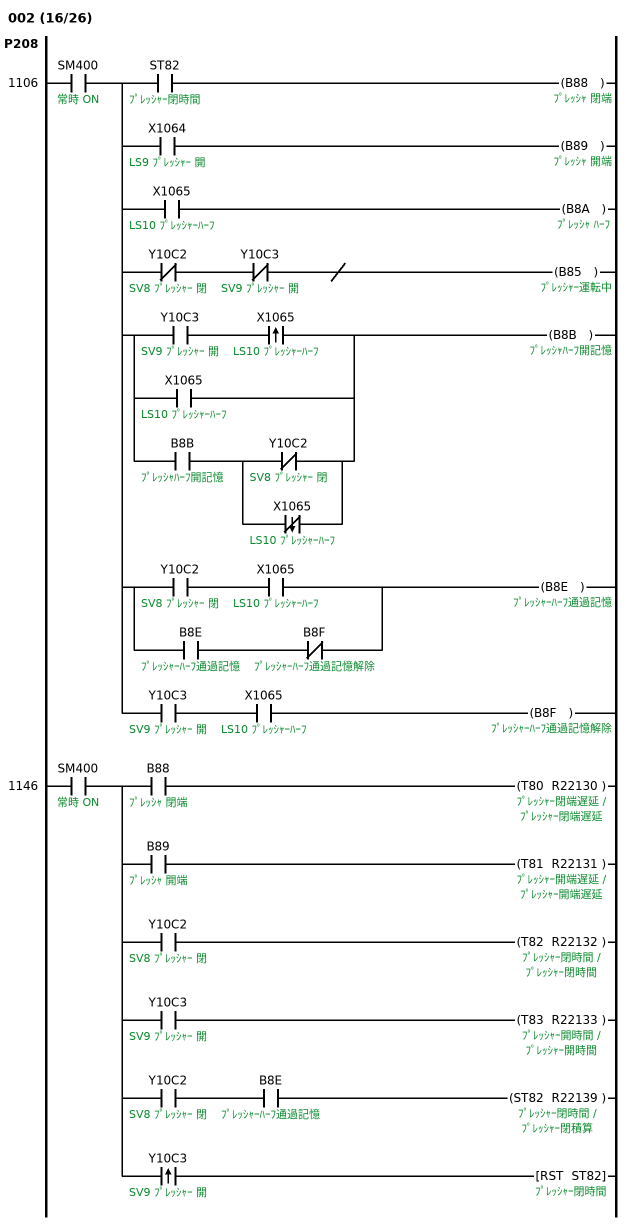
1106  LD      SM400  ; 常時 ON
      MPS
      AND     ST82  ; ﾌﾟﾚｯｼｬｰ閉時間
      OUT     B88  ; ﾌﾟﾚｯｼｬ 閉端
      MRD
      AND     X1064  ; LS9 ﾌﾟﾚｯｼｬｰ 開
      OUT     B89  ; ﾌﾟﾚｯｼｬ 開端
      MRD
      AND     X1065  ; LS10 ﾌﾟﾚｯｼｬｰﾊｰﾌ
      OUT     B8A  ; ﾌﾟﾚｯｼｬ ﾊｰﾌ
      MRD
      ANI     Y10C2  ; SV8 ﾌﾟﾚｯｼｬｰ 閉
      ANI     Y10C3  ; SV9 ﾌﾟﾚｯｼｬｰ 開
      INV
      OUT     B85  ; ﾌﾟﾚｯｼｬｰ運転中
      MRD
      LD      Y10C3  ; SV9 ﾌﾟﾚｯｼｬｰ 開
      ANDP    X1065  ; LS10 ﾌﾟﾚｯｼｬｰﾊｰﾌ
      OR      X1065  ; LS10 ﾌﾟﾚｯｼｬｰﾊｰﾌ
      LD      B8B  ; ﾌﾟﾚｯｼｬﾊｰﾌ開記憶
      LDI     Y10C2  ; SV8 ﾌﾟﾚｯｼｬｰ 閉
      ORFI    X1065  ; LS10 ﾌﾟﾚｯｼｬｰﾊｰﾌ
      ANB
      ORB
      ANB
      OUT     B8B  ; ﾌﾟﾚｯｼｬﾊｰﾌ開記憶
      MRD
      LD      Y10C2  ; SV8 ﾌﾟﾚｯｼｬｰ 閉
      AND     X1065  ; LS10 ﾌﾟﾚｯｼｬｰﾊｰﾌ
      LD      B8E  ; ﾌﾟﾚｯｼｬｰﾊｰﾌ通過記憶
      ANI     B8F  ; ﾌﾟﾚｯｼｬｰﾊｰﾌ通過記憶解除
      ORB
      ANB
      OUT     B8E  ; ﾌﾟﾚｯｼｬｰﾊｰﾌ通過記憶
      MPP
      AND     Y10C3  ; SV9 ﾌﾟﾚｯｼｬｰ 開
      AND     X1065  ; LS10 ﾌﾟﾚｯｼｬｰﾊｰﾌ
      OUT     B8F  ; ﾌﾟﾚｯｼｬｰﾊｰﾌ通過記憶解除
1146  LD      SM400  ; 常時 ON
      MPS
      AND     B88  ; ﾌﾟﾚｯｼｬ 閉端
      OUT     T80 R22130  ; ﾌﾟﾚｯｼｬｰ閉端遅延 / ﾌﾟﾚｯｼｬｰ閉端遅延
      MRD
      AND     B89  ; ﾌﾟﾚｯｼｬ 開端
      OUT     T81 R22131  ; ﾌﾟﾚｯｼｬｰ開端遅延 / ﾌﾟﾚｯｼｬｰ開端遅延
      MRD
      AND     Y10C2  ; SV8 ﾌﾟﾚｯｼｬｰ 閉
      OUT     T82 R22132  ; ﾌﾟﾚｯｼｬｰ閉時間 / ﾌﾟﾚｯｼｬｰ閉時間
      MRD
      AND     Y10C3  ; SV9 ﾌﾟﾚｯｼｬｰ 開
      OUT     T83 R22133  ; ﾌﾟﾚｯｼｬｰ開時間 / ﾌﾟﾚｯｼｬｰ開時間
      MRD
      AND     Y10C2  ; SV8 ﾌﾟﾚｯｼｬｰ 閉
      AND     B8E  ; ﾌﾟﾚｯｼｬｰﾊｰﾌ通過記憶
      OUT     ST82 R22139  ; ﾌﾟﾚｯｼｬｰ閉時間 / ﾌﾟﾚｯｼｬｰ閉積算
      MPP
      ANDP    Y10C3  ; SV9 ﾌﾟﾚｯｼｬｰ 開
      RST     ST82  ; ﾌﾟﾚｯｼｬｰ閉時間
; 
      P209
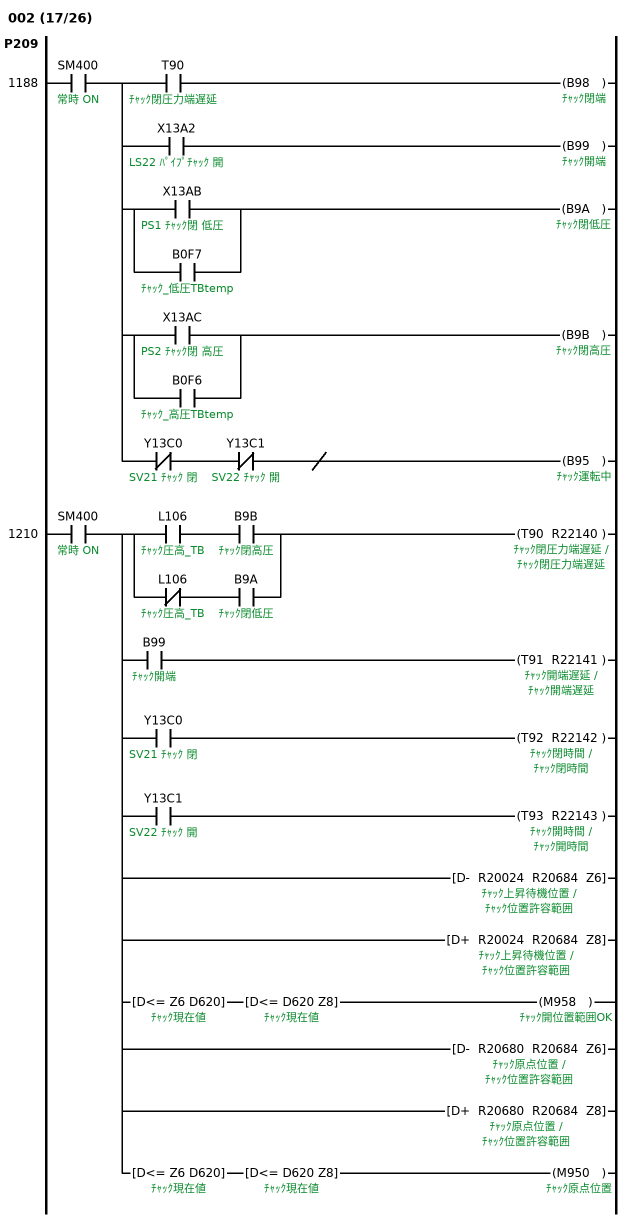
1188  LD      SM400  ; 常時 ON
      MPS
      AND     T90  ; ﾁｬｯｸ閉圧力端遅延
      OUT     B98  ; ﾁｬｯｸ閉端
      MRD
      AND     X13A2  ; LS22 ﾊﾟｲﾌﾟﾁｬｯｸ 開
      OUT     B99  ; ﾁｬｯｸ開端
      MRD
      LD      X13AB  ; PS1 ﾁｬｯｸ閉 低圧
      OR      B0F7  ; ﾁｬｯｸ_低圧TBtemp
      ANB
      OUT     B9A  ; ﾁｬｯｸ閉低圧
      MRD
      LD      X13AC  ; PS2 ﾁｬｯｸ閉 高圧
      OR      B0F6  ; ﾁｬｯｸ_高圧TBtemp
      ANB
      OUT     B9B  ; ﾁｬｯｸ閉高圧
      MPP
      ANI     Y13C0  ; SV21 ﾁｬｯｸ 閉
      ANI     Y13C1  ; SV22 ﾁｬｯｸ 開
      INV
      OUT     B95  ; ﾁｬｯｸ運転中
1210  LD      SM400  ; 常時 ON
      MPS
      LD      L106  ; ﾁｬｯｸ圧高_TB
      AND     B9B  ; ﾁｬｯｸ閉高圧
      LDI     L106  ; ﾁｬｯｸ圧高_TB
      AND     B9A  ; ﾁｬｯｸ閉低圧
      ORB
      ANB
      OUT     T90 R22140  ; ﾁｬｯｸ閉圧力端遅延 / ﾁｬｯｸ閉圧力端遅延
      MRD
      AND     B99  ; ﾁｬｯｸ開端
      OUT     T91 R22141  ; ﾁｬｯｸ開端遅延 / ﾁｬｯｸ開端遅延
      MRD
      AND     Y13C0  ; SV21 ﾁｬｯｸ 閉
      OUT     T92 R22142  ; ﾁｬｯｸ閉時間 / ﾁｬｯｸ閉時間
      MRD
      AND     Y13C1  ; SV22 ﾁｬｯｸ 開
      OUT     T93 R22143  ; ﾁｬｯｸ開時間 / ﾁｬｯｸ開時間
      MPP
      D-      R20024 R20684 Z6  ; ﾁｬｯｸ位置許容範囲
      D+      R20024 R20684 Z8
      MPS
      ANDD<=  Z6 D620  ; ﾁｬｯｸ現在値
      ANDD<=  D620 Z8  ; ﾁｬｯｸ現在値
      OUT     M958  ; ﾁｬｯｸ開位置範囲OK
      MPP
      D-      R20680 R20684 Z6  ; ﾁｬｯｸ原点位置
      D+      R20680 R20684 Z8
      ANDD<=  Z6 D620  ; ﾁｬｯｸ現在値
      ANDD<=  D620 Z8  ; ﾁｬｯｸ現在値
      OUT     M950  ; ﾁｬｯｸ原点位置
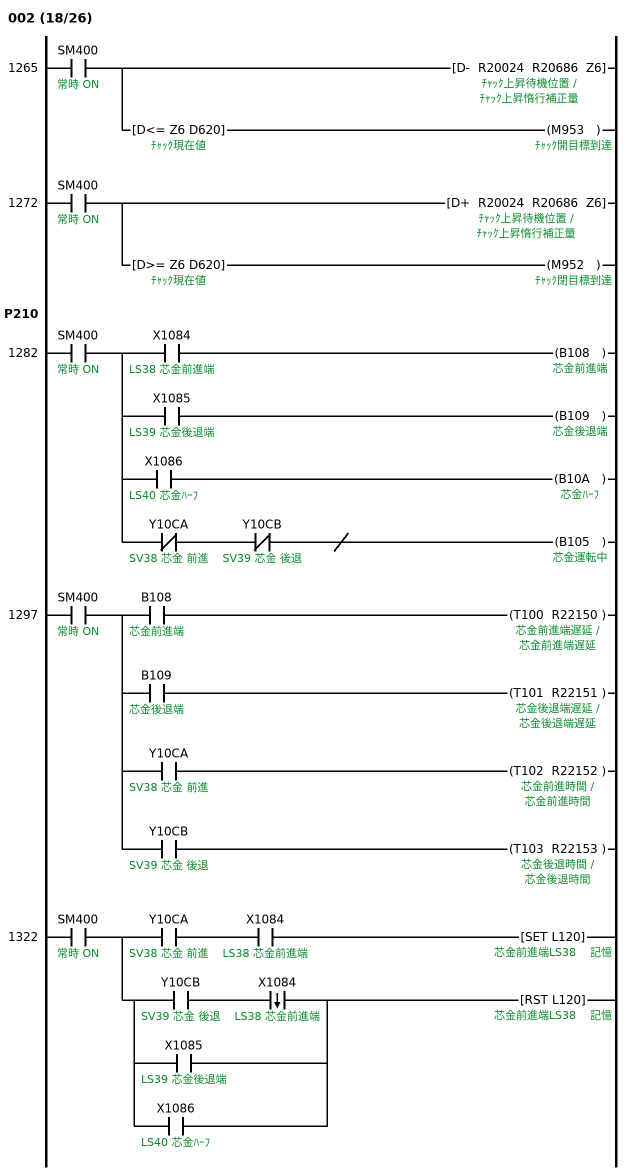
1265  LD      SM400  ; 常時 ON
      D-      R20024 R20686 Z6  ; ﾁｬｯｸ上昇惰行補正量
      ANDD<=  Z6 D620  ; ﾁｬｯｸ現在値
      OUT     M953  ; ﾁｬｯｸ開目標到達
1272  LD      SM400  ; 常時 ON
      D+      R20024 R20686 Z6
      ANDD>=  Z6 D620  ; ﾁｬｯｸ現在値
      OUT     M952  ; ﾁｬｯｸ閉目標到達
; 
      P210
1282  LD      SM400  ; 常時 ON
      MPS
      AND     X1084  ; LS38 芯金前進端
      OUT     B108  ; 芯金前進端
      MRD
      AND     X1085  ; LS39 芯金後退端
      OUT     B109  ; 芯金後退端
      MRD
      AND     X1086  ; LS40 芯金ﾊｰﾌ
      OUT     B10A  ; 芯金ﾊｰﾌ
      MPP
      ANI     Y10CA  ; SV38 芯金 前進
      ANI     Y10CB  ; SV39 芯金 後退
      INV
      OUT     B105  ; 芯金運転中
1297  LD      SM400  ; 常時 ON
      MPS
      AND     B108  ; 芯金前進端
      OUT     T100 R22150  ; 芯金前進端遅延 / 芯金前進端遅延
      MRD
      AND     B109  ; 芯金後退端
      OUT     T101 R22151  ; 芯金後退端遅延 / 芯金後退端遅延
      MRD
      AND     Y10CA  ; SV38 芯金 前進
      OUT     T102 R22152  ; 芯金前進時間 / 芯金前進時間
      MPP
      AND     Y10CB  ; SV39 芯金 後退
      OUT     T103 R22153  ; 芯金後退時間 / 芯金後退時間
1322  LD      SM400  ; 常時 ON
      MPS
      AND     Y10CA  ; SV38 芯金 前進
      AND     X1084  ; LS38 芯金前進端
      SET     L120  ; 芯金前進端LS38    記憶
      MPP
      LD      Y10CB  ; SV39 芯金 後退
      ANDF    X1084  ; LS38 芯金前進端
      OR      X1085  ; LS39 芯金後退端
      OR      X1086  ; LS40 芯金ﾊｰﾌ
      ANB
      RST     L120  ; 芯金前進端LS38    記憶
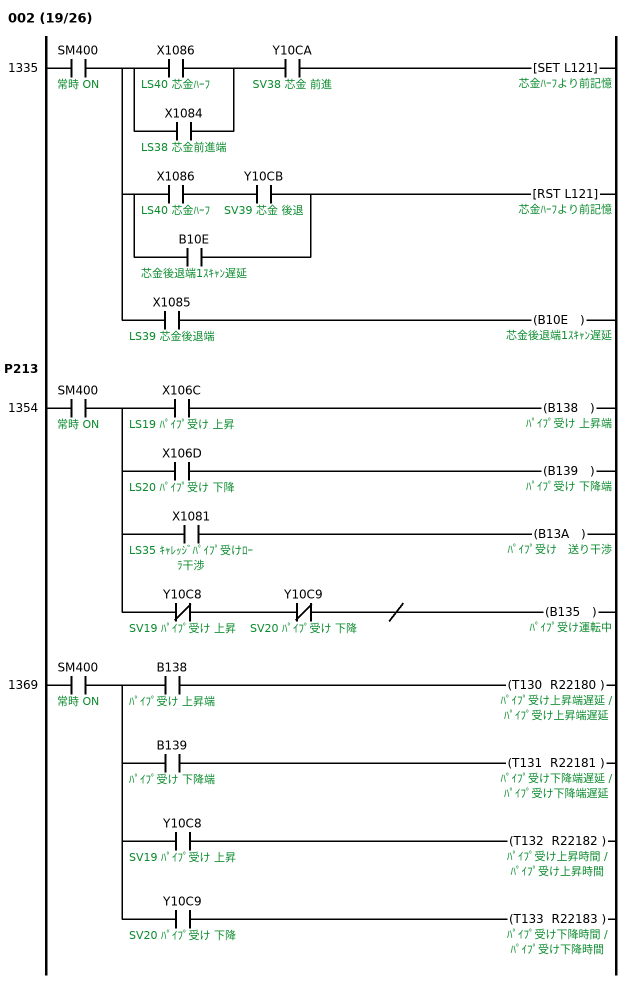
1335  LD      SM400  ; 常時 ON
      MPS
      LD      X1086  ; LS40 芯金ﾊｰﾌ
      OR      X1084  ; LS38 芯金前進端
      ANB
      AND     Y10CA  ; SV38 芯金 前進
      SET     L121  ; 芯金ﾊｰﾌより前記憶
      MRD
      LD      X1086  ; LS40 芯金ﾊｰﾌ
      AND     Y10CB  ; SV39 芯金 後退
      OR      B10E  ; 芯金後退端1ｽｷｬﾝ遅延
      ANB
      RST     L121  ; 芯金ﾊｰﾌより前記憶
      MPP
      AND     X1085  ; LS39 芯金後退端
      OUT     B10E  ; 芯金後退端1ｽｷｬﾝ遅延
; 
      P213
1354  LD      SM400  ; 常時 ON
      MPS
      AND     X106C  ; LS19 ﾊﾟｲﾌﾟ受け 上昇
      OUT     B138  ; ﾊﾟｲﾌﾟ受け 上昇端
      MRD
      AND     X106D  ; LS20 ﾊﾟｲﾌﾟ受け 下降
      OUT     B139  ; ﾊﾟｲﾌﾟ受け 下降端
      MRD
      AND     X1081  ; LS35 ｷｬﾚｯｼﾞﾊﾟｲﾌﾟ受けﾛｰﾗ干渉
      OUT     B13A  ; ﾊﾟｲﾌﾟ受け　送り干渉
      MPP
      ANI     Y10C8  ; SV19 ﾊﾟｲﾌﾟ受け 上昇
      ANI     Y10C9  ; SV20 ﾊﾟｲﾌﾟ受け 下降
      INV
      OUT     B135  ; ﾊﾟｲﾌﾟ受け運転中
1369  LD      SM400  ; 常時 ON
      MPS
      AND     B138  ; ﾊﾟｲﾌﾟ受け 上昇端
      OUT     T130 R22180  ; ﾊﾟｲﾌﾟ受け上昇端遅延 / ﾊﾟｲﾌﾟ受け上昇端遅延
      MRD
      AND     B139  ; ﾊﾟｲﾌﾟ受け 下降端
      OUT     T131 R22181  ; ﾊﾟｲﾌﾟ受け下降端遅延 / ﾊﾟｲﾌﾟ受け下降端遅延
      MRD
      AND     Y10C8  ; SV19 ﾊﾟｲﾌﾟ受け 上昇
      OUT     T132 R22182  ; ﾊﾟｲﾌﾟ受け上昇時間 / ﾊﾟｲﾌﾟ受け上昇時間
      MPP
      AND     Y10C9  ; SV20 ﾊﾟｲﾌﾟ受け 下降
      OUT     T133 R22183  ; ﾊﾟｲﾌﾟ受け下降時間 / ﾊﾟｲﾌﾟ受け下降時間
; 
      P214
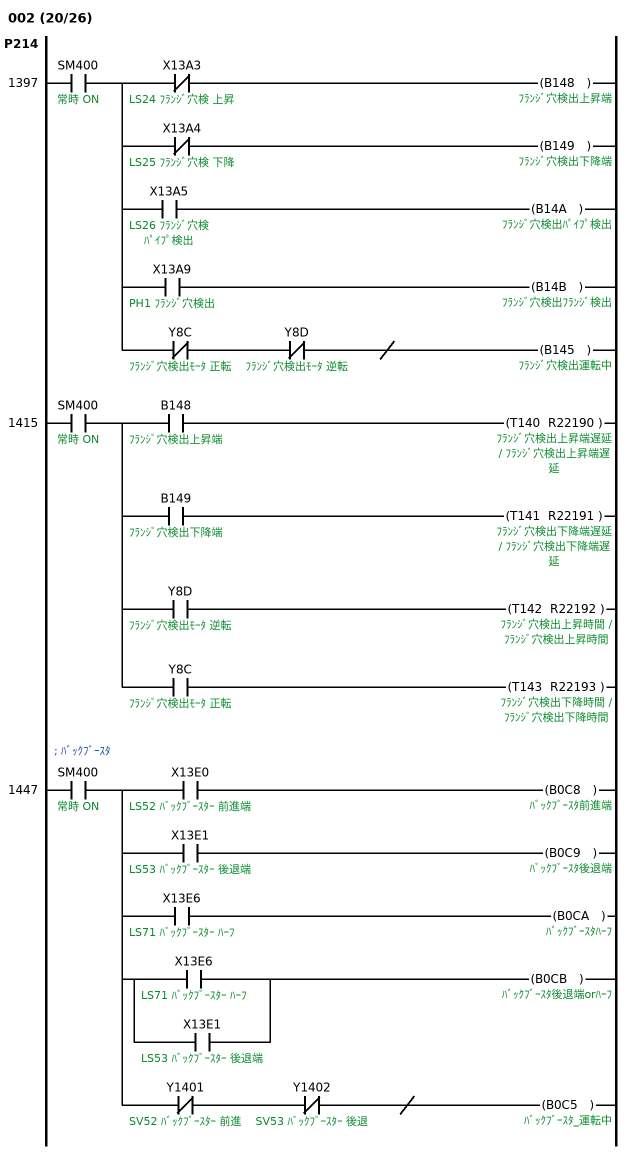
1397  LD      SM400  ; 常時 ON
      MPS
      ANI     X13A3  ; LS24 ﾌﾗﾝｼﾞ穴検 上昇
      OUT     B148  ; ﾌﾗﾝｼﾞ穴検出上昇端
      MRD
      ANI     X13A4  ; LS25 ﾌﾗﾝｼﾞ穴検 下降
      OUT     B149  ; ﾌﾗﾝｼﾞ穴検出下降端
      MRD
      AND     X13A5  ; LS26 ﾌﾗﾝｼﾞ穴検 ﾊﾟｲﾌﾟ検出
      OUT     B14A  ; ﾌﾗﾝｼﾞ穴検出ﾊﾟｲﾌﾟ検出
      MRD
      AND     X13A9  ; PH1 ﾌﾗﾝｼﾞ穴検出
      OUT     B14B  ; ﾌﾗﾝｼﾞ穴検出ﾌﾗﾝｼﾞ検出
      MPP
      ANI     Y8C  ; ﾌﾗﾝｼﾞ穴検出ﾓｰﾀ 正転
      ANI     Y8D  ; ﾌﾗﾝｼﾞ穴検出ﾓｰﾀ 逆転
      INV
      OUT     B145  ; ﾌﾗﾝｼﾞ穴検出運転中
1415  LD      SM400  ; 常時 ON
      MPS
      AND     B148  ; ﾌﾗﾝｼﾞ穴検出上昇端
      OUT     T140 R22190  ; ﾌﾗﾝｼﾞ穴検出上昇端遅延 / ﾌﾗﾝｼﾞ穴検出上昇端遅延
      MRD
      AND     B149  ; ﾌﾗﾝｼﾞ穴検出下降端
      OUT     T141 R22191  ; ﾌﾗﾝｼﾞ穴検出下降端遅延 / ﾌﾗﾝｼﾞ穴検出下降端遅延
      MRD
      AND     Y8D  ; ﾌﾗﾝｼﾞ穴検出ﾓｰﾀ 逆転
      OUT     T142 R22192  ; ﾌﾗﾝｼﾞ穴検出上昇時間 / ﾌﾗﾝｼﾞ穴検出上昇時間
      MPP
      AND     Y8C  ; ﾌﾗﾝｼﾞ穴検出ﾓｰﾀ 正転
      OUT     T143 R22193  ; ﾌﾗﾝｼﾞ穴検出下降時間 / ﾌﾗﾝｼﾞ穴検出下降時間
; ﾊﾞｯｸﾌﾞｰｽﾀ
1447  LD      SM400  ; 常時 ON
      MPS
      AND     X13E0  ; LS52 ﾊﾞｯｸﾌﾞｰｽﾀｰ 前進端
      OUT     B0C8  ; ﾊﾞｯｸﾌﾞｰｽﾀ前進端
      MRD
      AND     X13E1  ; LS53 ﾊﾞｯｸﾌﾞｰｽﾀｰ 後退端
      OUT     B0C9  ; ﾊﾞｯｸﾌﾞｰｽﾀ後退端
      MRD
      AND     X13E6  ; LS71 ﾊﾞｯｸﾌﾞｰｽﾀｰ ﾊｰﾌ
      OUT     B0CA  ; ﾊﾞｯｸﾌﾞｰｽﾀﾊｰﾌ
      MRD
      LD      X13E6  ; LS71 ﾊﾞｯｸﾌﾞｰｽﾀｰ ﾊｰﾌ
      OR      X13E1  ; LS53 ﾊﾞｯｸﾌﾞｰｽﾀｰ 後退端
      ANB
      OUT     B0CB  ; ﾊﾞｯｸﾌﾞｰｽﾀ後退端orﾊｰﾌ
      MPP
      ANI     Y1401  ; SV52 ﾊﾞｯｸﾌﾞｰｽﾀｰ 前進
      ANI     Y1402  ; SV53 ﾊﾞｯｸﾌﾞｰｽﾀｰ 後退
      INV
      OUT     B0C5  ; ﾊﾞｯｸﾌﾞｰｽﾀ_運転中
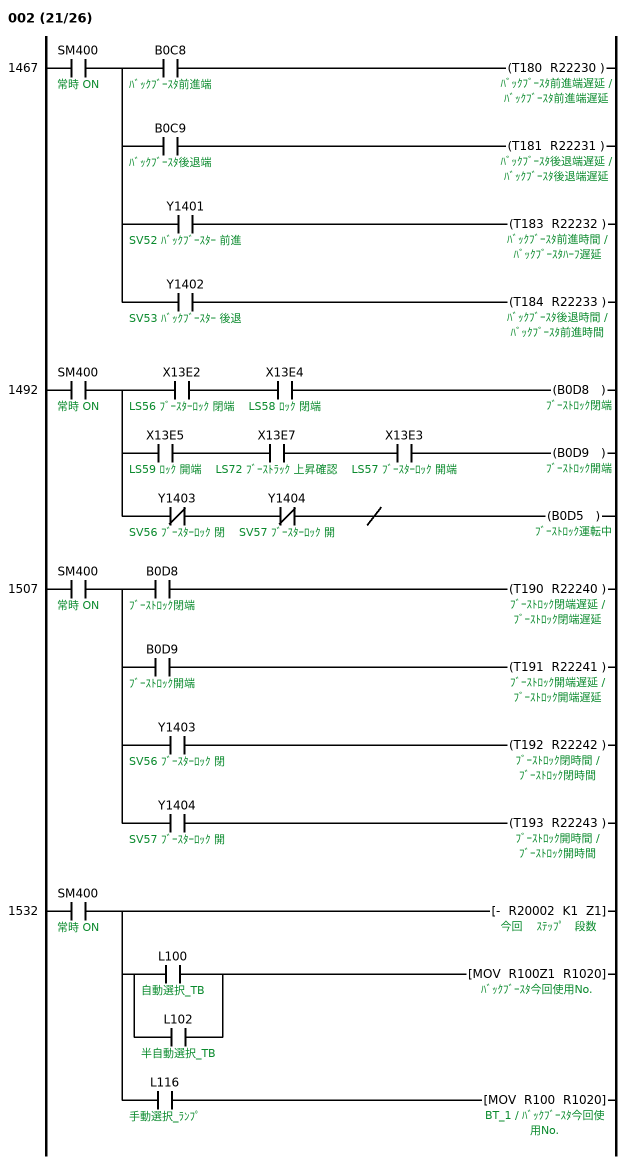
1467  LD      SM400  ; 常時 ON
      MPS
      AND     B0C8  ; ﾊﾞｯｸﾌﾞｰｽﾀ前進端
      OUT     T180 R22230  ; ﾊﾞｯｸﾌﾞｰｽﾀ前進端遅延 / ﾊﾞｯｸﾌﾞｰｽﾀ前進端遅延
      MRD
      AND     B0C9  ; ﾊﾞｯｸﾌﾞｰｽﾀ後退端
      OUT     T181 R22231  ; ﾊﾞｯｸﾌﾞｰｽﾀ後退端遅延 / ﾊﾞｯｸﾌﾞｰｽﾀ後退端遅延
      MRD
      AND     Y1401  ; SV52 ﾊﾞｯｸﾌﾞｰｽﾀｰ 前進
      OUT     T183 R22232  ; ﾊﾞｯｸﾌﾞｰｽﾀ前進時間 / ﾊﾞｯｸﾌﾞｰｽﾀﾊｰﾌ遅延
      MPP
      AND     Y1402  ; SV53 ﾊﾞｯｸﾌﾞｰｽﾀｰ 後退
      OUT     T184 R22233  ; ﾊﾞｯｸﾌﾞｰｽﾀ後退時間 / ﾊﾞｯｸﾌﾞｰｽﾀ前進時間
1492  LD      SM400  ; 常時 ON
      MPS
      AND     X13E2  ; LS56 ﾌﾞｰｽﾀｰﾛｯｸ 閉端
      AND     X13E4  ; LS58 ﾛｯｸ 閉端
      OUT     B0D8  ; ﾌﾞｰｽﾄﾛｯｸ閉端
      MRD
      AND     X13E5  ; LS59 ﾛｯｸ 開端
      AND     X13E7  ; LS72 ﾌﾞｰｽﾄﾗｯｸ 上昇確認
      AND     X13E3  ; LS57 ﾌﾞｰｽﾀｰﾛｯｸ 開端
      OUT     B0D9  ; ﾌﾞｰｽﾄﾛｯｸ開端
      MPP
      ANI     Y1403  ; SV56 ﾌﾞｰｽﾀｰﾛｯｸ 閉
      ANI     Y1404  ; SV57 ﾌﾞｰｽﾀｰﾛｯｸ 開
      INV
      OUT     B0D5  ; ﾌﾞｰｽﾄﾛｯｸ運転中
1507  LD      SM400  ; 常時 ON
      MPS
      AND     B0D8  ; ﾌﾞｰｽﾄﾛｯｸ閉端
      OUT     T190 R22240  ; ﾌﾞｰｽﾄﾛｯｸ閉端遅延 / ﾌﾞｰｽﾄﾛｯｸ閉端遅延
      MRD
      AND     B0D9  ; ﾌﾞｰｽﾄﾛｯｸ開端
      OUT     T191 R22241  ; ﾌﾞｰｽﾄﾛｯｸ開端遅延 / ﾌﾞｰｽﾄﾛｯｸ開端遅延
      MRD
      AND     Y1403  ; SV56 ﾌﾞｰｽﾀｰﾛｯｸ 閉
      OUT     T192 R22242  ; ﾌﾞｰｽﾄﾛｯｸ閉時間 / ﾌﾞｰｽﾄﾛｯｸ閉時間
      MPP
      AND     Y1404  ; SV57 ﾌﾞｰｽﾀｰﾛｯｸ 開
      OUT     T193 R22243  ; ﾌﾞｰｽﾄﾛｯｸ開時間 / ﾌﾞｰｽﾄﾛｯｸ開時間
1532  LD      SM400  ; 常時 ON
      -       R20002 K1 Z1  ; 今回    ｽﾃｯﾌﾟ   段数
      MPS
      LD      L100  ; 自動選択_TB
      OR      L102  ; 半自動選択_TB
      ANB
      MOV     R100Z1 R1020  ; ﾊﾞｯｸﾌﾞｰｽﾀ今回使用No.
      MPP
      AND     L116  ; 手動選択_ﾗﾝﾌﾟ
      MOV     R100 R1020  ; BT_1
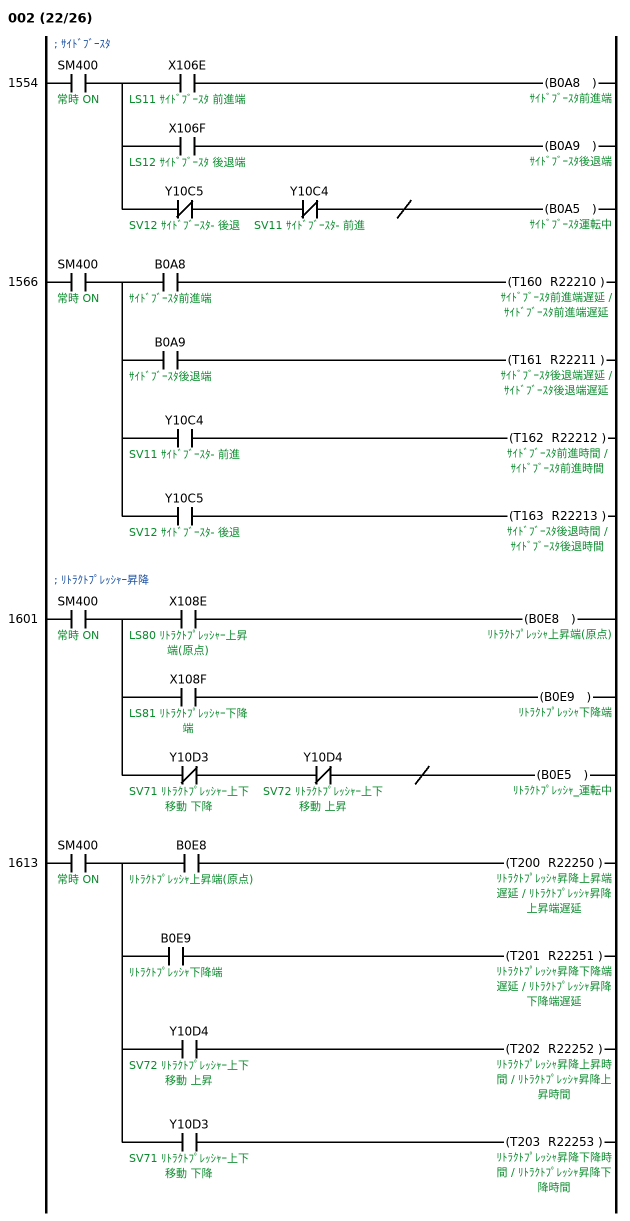
; ｻｲﾄﾞﾌﾞｰｽﾀ
1554  LD      SM400  ; 常時 ON
      MPS
      AND     X106E  ; LS11 ｻｲﾄﾞﾌﾞｰｽﾀ 前進端
      OUT     B0A8  ; ｻｲﾄﾞﾌﾞｰｽﾀ前進端
      MRD
      AND     X106F  ; LS12 ｻｲﾄﾞﾌﾞｰｽﾀ 後退端
      OUT     B0A9  ; ｻｲﾄﾞﾌﾞｰｽﾀ後退端
      MPP
      ANI     Y10C5  ; SV12 ｻｲﾄﾞﾌﾞｰｽﾀ- 後退
      ANI     Y10C4  ; SV11 ｻｲﾄﾞﾌﾞｰｽﾀ- 前進
      INV
      OUT     B0A5  ; ｻｲﾄﾞﾌﾞｰｽﾀ運転中
1566  LD      SM400  ; 常時 ON
      MPS
      AND     B0A8  ; ｻｲﾄﾞﾌﾞｰｽﾀ前進端
      OUT     T160 R22210  ; ｻｲﾄﾞﾌﾞｰｽﾀ前進端遅延 / ｻｲﾄﾞﾌﾞｰｽﾀ前進端遅延
      MRD
      AND     B0A9  ; ｻｲﾄﾞﾌﾞｰｽﾀ後退端
      OUT     T161 R22211  ; ｻｲﾄﾞﾌﾞｰｽﾀ後退端遅延 / ｻｲﾄﾞﾌﾞｰｽﾀ後退端遅延
      MRD
      AND     Y10C4  ; SV11 ｻｲﾄﾞﾌﾞｰｽﾀ- 前進
      OUT     T162 R22212  ; ｻｲﾄﾞﾌﾞｰｽﾀ前進時間 / ｻｲﾄﾞﾌﾞｰｽﾀ前進時間
      MPP
      AND     Y10C5  ; SV12 ｻｲﾄﾞﾌﾞｰｽﾀ- 後退
      OUT     T163 R22213  ; ｻｲﾄﾞﾌﾞｰｽﾀ後退時間 / ｻｲﾄﾞﾌﾞｰｽﾀ後退時間
; ﾘﾄﾗｸﾄﾌﾟﾚｯｼｬｰ昇降
1601  LD      SM400  ; 常時 ON
      MPS
      AND     X108E  ; LS80 ﾘﾄﾗｸﾄﾌﾟﾚｯｼｬｰ上昇端(原点)
      OUT     B0E8  ; ﾘﾄﾗｸﾄﾌﾟﾚｯｼｬ上昇端(原点)
      MRD
      AND     X108F  ; LS81 ﾘﾄﾗｸﾄﾌﾟﾚｯｼｬｰ下降端
      OUT     B0E9  ; ﾘﾄﾗｸﾄﾌﾟﾚｯｼｬ下降端
      MPP
      ANI     Y10D3  ; SV71 ﾘﾄﾗｸﾄﾌﾟﾚｯｼｬｰ上下移動 下降
      ANI     Y10D4  ; SV72 ﾘﾄﾗｸﾄﾌﾟﾚｯｼｬｰ上下移動 上昇
      INV
      OUT     B0E5  ; ﾘﾄﾗｸﾄﾌﾟﾚｯｼｬ_運転中
1613  LD      SM400  ; 常時 ON
      MPS
      AND     B0E8  ; ﾘﾄﾗｸﾄﾌﾟﾚｯｼｬ上昇端(原点)
      OUT     T200 R22250  ; ﾘﾄﾗｸﾄﾌﾟﾚｯｼｬ昇降上昇端遅延 / ﾘﾄﾗｸﾄﾌﾟﾚｯｼｬ昇降上昇端遅延
      MRD
      AND     B0E9  ; ﾘﾄﾗｸﾄﾌﾟﾚｯｼｬ下降端
      OUT     T201 R22251  ; ﾘﾄﾗｸﾄﾌﾟﾚｯｼｬ昇降下降端遅延 / ﾘﾄﾗｸﾄﾌﾟﾚｯｼｬ昇降下降端遅延
      MRD
      AND     Y10D4  ; SV72 ﾘﾄﾗｸﾄﾌﾟﾚｯｼｬｰ上下移動 上昇
      OUT     T202 R22252  ; ﾘﾄﾗｸﾄﾌﾟﾚｯｼｬ昇降上昇時間 / ﾘﾄﾗｸﾄﾌﾟﾚｯｼｬ昇降上昇時間
      MPP
      AND     Y10D3  ; SV71 ﾘﾄﾗｸﾄﾌﾟﾚｯｼｬｰ上下移動 下降
      OUT     T203 R22253  ; ﾘﾄﾗｸﾄﾌﾟﾚｯｼｬ昇降下降時間 / ﾘﾄﾗｸﾄﾌﾟﾚｯｼｬ昇降下降時間
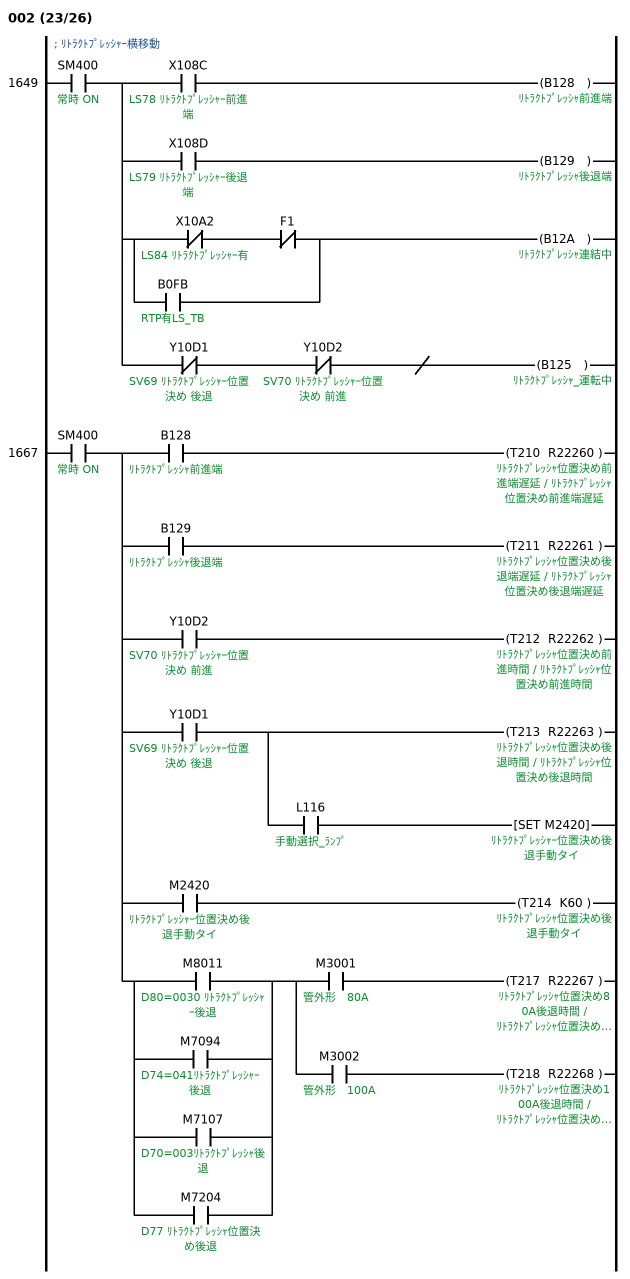
; ﾘﾄﾗｸﾄﾌﾟﾚｯｼｬｰ横移動
1649  LD      SM400  ; 常時 ON
      MPS
      AND     X108C  ; LS78 ﾘﾄﾗｸﾄﾌﾟﾚｯｼｬｰ前進端
      OUT     B128  ; ﾘﾄﾗｸﾄﾌﾟﾚｯｼｬ前進端
      MRD
      AND     X108D  ; LS79 ﾘﾄﾗｸﾄﾌﾟﾚｯｼｬｰ後退端
      OUT     B129  ; ﾘﾄﾗｸﾄﾌﾟﾚｯｼｬ後退端
      MRD
      LDI     X10A2  ; LS84 ﾘﾄﾗｸﾄﾌﾟﾚｯｼｬｰ有
      ANI     F1
      OR      B0FB  ; RTP有LS_TB
      ANB
      OUT     B12A  ; ﾘﾄﾗｸﾄﾌﾟﾚｯｼｬ連結中
      MPP
      ANI     Y10D1  ; SV69 ﾘﾄﾗｸﾄﾌﾟﾚｯｼｬｰ位置決め 後退
      ANI     Y10D2  ; SV70 ﾘﾄﾗｸﾄﾌﾟﾚｯｼｬｰ位置決め 前進
      INV
      OUT     B125  ; ﾘﾄﾗｸﾄﾌﾟﾚｯｼｬ_運転中
1667  LD      SM400  ; 常時 ON
      MPS
      AND     B128  ; ﾘﾄﾗｸﾄﾌﾟﾚｯｼｬ前進端
      OUT     T210 R22260  ; ﾘﾄﾗｸﾄﾌﾟﾚｯｼｬ位置決め前進端遅延 / ﾘﾄﾗｸﾄﾌﾟﾚｯｼｬ位置決め前進端遅延
      MRD
      AND     B129  ; ﾘﾄﾗｸﾄﾌﾟﾚｯｼｬ後退端
      OUT     T211 R22261  ; ﾘﾄﾗｸﾄﾌﾟﾚｯｼｬ位置決め後退端遅延 / ﾘﾄﾗｸﾄﾌﾟﾚｯｼｬ位置決め後退端遅延
      MRD
      AND     Y10D2  ; SV70 ﾘﾄﾗｸﾄﾌﾟﾚｯｼｬｰ位置決め 前進
      OUT     T212 R22262  ; ﾘﾄﾗｸﾄﾌﾟﾚｯｼｬ位置決め前進時間 / ﾘﾄﾗｸﾄﾌﾟﾚｯｼｬ位置決め前進時間
      MRD
      AND     Y10D1  ; SV69 ﾘﾄﾗｸﾄﾌﾟﾚｯｼｬｰ位置決め 後退
      OUT     T213 R22263  ; ﾘﾄﾗｸﾄﾌﾟﾚｯｼｬ位置決め後退時間 / ﾘﾄﾗｸﾄﾌﾟﾚｯｼｬ位置決め後退時間
      AND     L116  ; 手動選択_ﾗﾝﾌﾟ
      SET     M2420  ; ﾘﾄﾗｸﾄﾌﾟﾚｯｼｬｰ位置決め後退手動タイ
      MRD
      AND     M2420  ; ﾘﾄﾗｸﾄﾌﾟﾚｯｼｬｰ位置決め後退手動タイ
      OUT     T214 K60  ; ﾘﾄﾗｸﾄﾌﾟﾚｯｼｬ位置決め後退手動タイ
      MPP
      LD      M8011  ; D80=0030 ﾘﾄﾗｸﾄﾌﾟﾚｯｼｬｰ後退
      OR      M7094  ; D74=041ﾘﾄﾗｸﾄﾌﾟﾚｯｼｬｰ後退
      OR      M7107  ; D70=003ﾘﾄﾗｸﾄﾌﾟﾚｯｼｬ後退
      OR      M7204  ; D77 ﾘﾄﾗｸﾄﾌﾟﾚｯｼｬ位置決め後退
      ANB
      MPS
      AND     M3001  ; 管外形　80A
      OUT     T217 R22267  ; ﾘﾄﾗｸﾄﾌﾟﾚｯｼｬ位置決め80A後退時間 / ﾘﾄﾗｸﾄﾌﾟﾚｯｼｬ位置決め80A後退時間
      MPP
      AND     M3002  ; 管外形　100A
      OUT     T218 R22268  ; ﾘﾄﾗｸﾄﾌﾟﾚｯｼｬ位置決め100A後退時間 / ﾘﾄﾗｸﾄﾌﾟﾚｯｼｬ位置決め100A後退時間
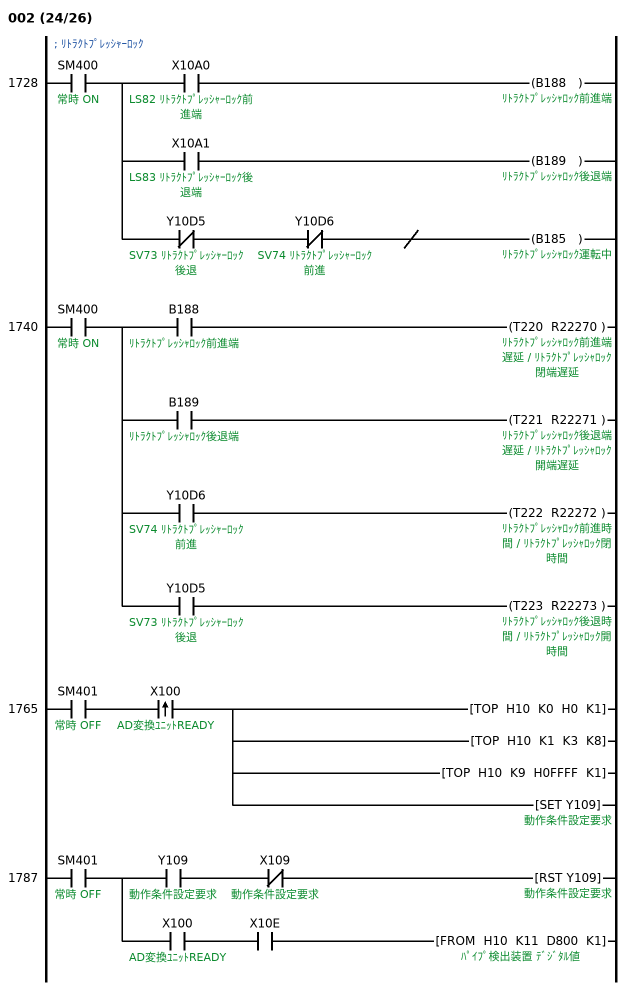
; ﾘﾄﾗｸﾄﾌﾟﾚｯｼｬｰﾛｯｸ
1728  LD      SM400  ; 常時 ON
      MPS
      AND     X10A0  ; LS82 ﾘﾄﾗｸﾄﾌﾟﾚｯｼｬｰﾛｯｸ前進端
      OUT     B188  ; ﾘﾄﾗｸﾄﾌﾟﾚｯｼｬﾛｯｸ前進端
      MRD
      AND     X10A1  ; LS83 ﾘﾄﾗｸﾄﾌﾟﾚｯｼｬｰﾛｯｸ後退端
      OUT     B189  ; ﾘﾄﾗｸﾄﾌﾟﾚｯｼｬﾛｯｸ後退端
      MPP
      ANI     Y10D5  ; SV73 ﾘﾄﾗｸﾄﾌﾟﾚｯｼｬｰﾛｯｸ 後退
      ANI     Y10D6  ; SV74 ﾘﾄﾗｸﾄﾌﾟﾚｯｼｬｰﾛｯｸ 前進
      INV
      OUT     B185  ; ﾘﾄﾗｸﾄﾌﾟﾚｯｼｬﾛｯｸ運転中
1740  LD      SM400  ; 常時 ON
      MPS
      AND     B188  ; ﾘﾄﾗｸﾄﾌﾟﾚｯｼｬﾛｯｸ前進端
      OUT     T220 R22270  ; ﾘﾄﾗｸﾄﾌﾟﾚｯｼｬﾛｯｸ前進端遅延 / ﾘﾄﾗｸﾄﾌﾟﾚｯｼｬﾛｯｸ閉端遅延
      MRD
      AND     B189  ; ﾘﾄﾗｸﾄﾌﾟﾚｯｼｬﾛｯｸ後退端
      OUT     T221 R22271  ; ﾘﾄﾗｸﾄﾌﾟﾚｯｼｬﾛｯｸ後退端遅延 / ﾘﾄﾗｸﾄﾌﾟﾚｯｼｬﾛｯｸ開端遅延
      MRD
      AND     Y10D6  ; SV74 ﾘﾄﾗｸﾄﾌﾟﾚｯｼｬｰﾛｯｸ 前進
      OUT     T222 R22272  ; ﾘﾄﾗｸﾄﾌﾟﾚｯｼｬﾛｯｸ前進時間 / ﾘﾄﾗｸﾄﾌﾟﾚｯｼｬﾛｯｸ閉時間
      MPP
      AND     Y10D5  ; SV73 ﾘﾄﾗｸﾄﾌﾟﾚｯｼｬｰﾛｯｸ 後退
      OUT     T223 R22273  ; ﾘﾄﾗｸﾄﾌﾟﾚｯｼｬﾛｯｸ後退時間 / ﾘﾄﾗｸﾄﾌﾟﾚｯｼｬﾛｯｸ開時間
1765  LD      SM401  ; 常時 OFF
      ANDP    X100  ; AD変換ﾕﾆｯﾄREADY
      TOP     H10 K0 H0 K1
      TOP     H10 K1 K3 K8
      TOP     H10 K9 H0FFFF K1
      SET     Y109  ; 動作条件設定要求
1787  LD      SM401  ; 常時 OFF
      MPS
      AND     Y109  ; 動作条件設定要求
      ANI     X109  ; 動作条件設定要求
      RST     Y109  ; 動作条件設定要求
      MPP
      AND     X100  ; AD変換ﾕﾆｯﾄREADY
      AND     X10E
      FROM    H10 K11 D800 K1  ; ﾊﾟｲﾌﾟ検出装置 ﾃﾞｼﾞﾀﾙ値
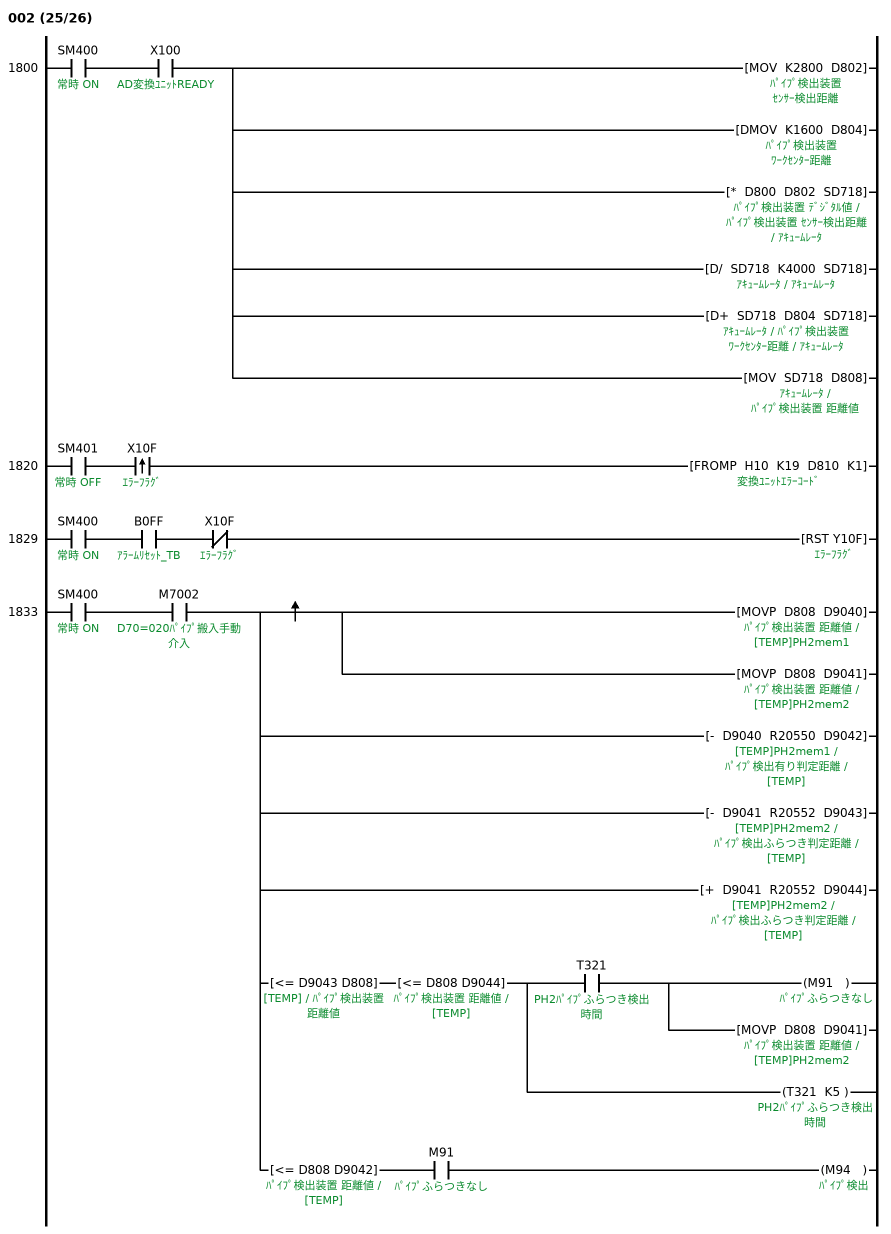
1800  LD      SM400  ; 常時 ON
      AND     X100  ; AD変換ﾕﾆｯﾄREADY
      MOV     K2800 D802  ; ﾊﾟｲﾌﾟ検出装置 ｾﾝｻｰ検出距離
      DMOV    K1600 D804  ; ﾊﾟｲﾌﾟ検出装置 ﾜｰｸｾﾝﾀｰ距離
      *       D800 D802 SD718  ; ｱｷｭｰﾑﾚｰﾀ
      D/      SD718 K4000 SD718
      D+      SD718 D804 SD718
      MOV     SD718 D808  ; ﾊﾟｲﾌﾟ検出装置 距離値
1820  LD      SM401  ; 常時 OFF
      ANDP    X10F  ; ｴﾗｰﾌﾗｸﾞ
      FROMP   H10 K19 D810 K1  ; 変換ﾕﾆｯﾄｴﾗｰｺｰﾄﾞ
1829  LD      SM400  ; 常時 ON
      AND     B0FF  ; ｱﾗｰﾑﾘｾｯﾄ_TB
      ANI     X10F  ; ｴﾗｰﾌﾗｸﾞ
      RST     Y10F  ; ｴﾗｰﾌﾗｸﾞ
1833  LD      SM400  ; 常時 ON
      AND     M7002  ; D70=020ﾊﾟｲﾌﾟ搬入手動介入
      MPS
      MEP
      MOVP    D808 D9040  ; [TEMP]PH2mem1
      MOVP    D808 D9041  ; [TEMP]PH2mem2
      MPP
      -       D9040 R20550 D9042  ; ﾊﾟｲﾌﾟ検出有り判定距離 / [TEMP]
      -       D9041 R20552 D9043  ; ﾊﾟｲﾌﾟ検出ふらつき判定距離 / [TEMP]
      +       D9041 R20552 D9044  ; [TEMP]
      MPS
      AND<=   D9043 D808  ; [TEMP] / ﾊﾟｲﾌﾟ検出装置 距離値
      AND<=   D808 D9044  ; ﾊﾟｲﾌﾟ検出装置 距離値 / [TEMP]
      MPS
      AND     T321  ; PH2ﾊﾟｲﾌﾟふらつき検出時間
      OUT     M91  ; ﾊﾟｲﾌﾟふらつきなし
      MOVP    D808 D9041
      MPP
      OUT     T321 K5  ; PH2ﾊﾟｲﾌﾟふらつき検出時間
      MPP
      AND<=   D808 D9042  ; ﾊﾟｲﾌﾟ検出装置 距離値 / [TEMP]
      AND     M91  ; ﾊﾟｲﾌﾟふらつきなし
      OUT     M94  ; ﾊﾟｲﾌﾟ検出
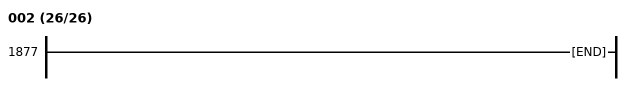
1877  END
END_PROGRAM

PROGRAM 003  // 異常
; 
      P300
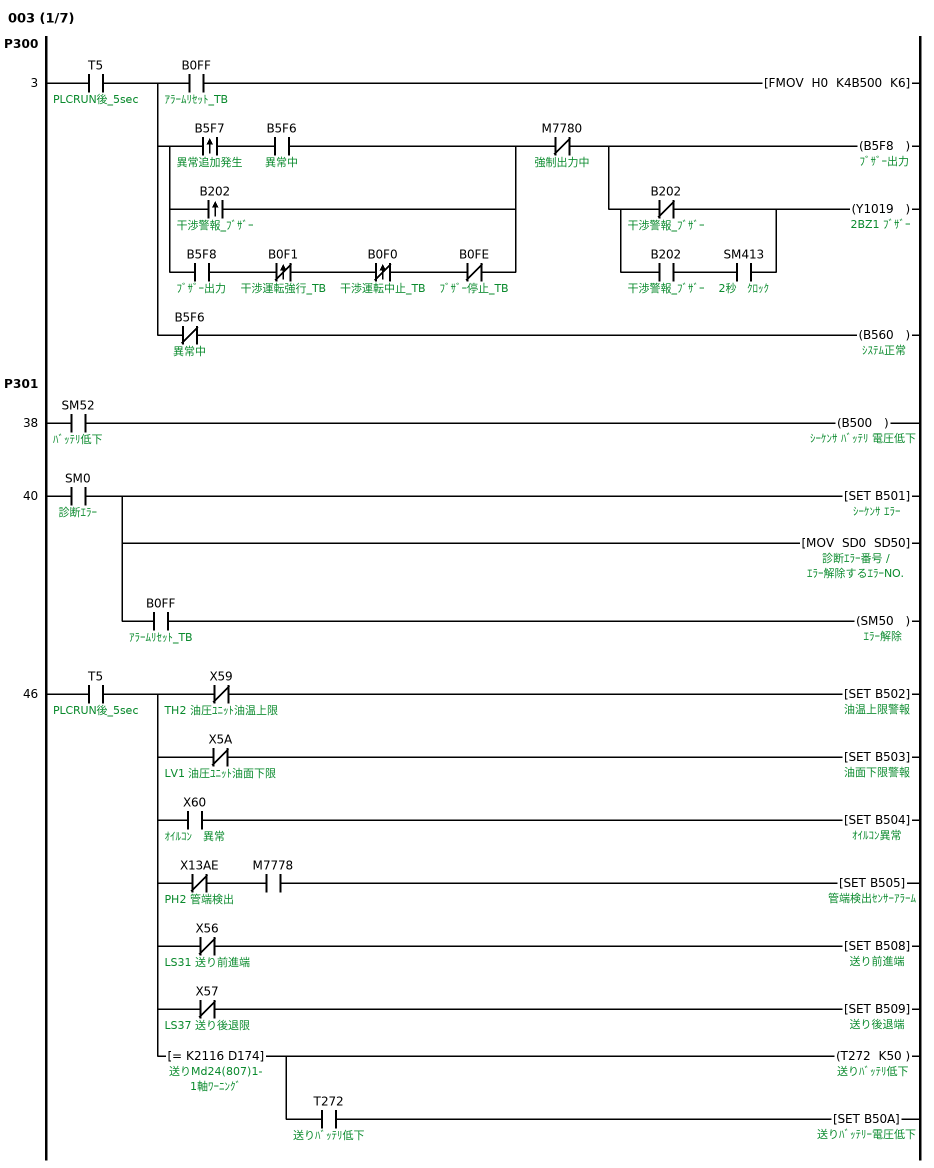
3     LD      T5  ; PLCRUN後_5sec
      MPS
      AND     B0FF  ; ｱﾗｰﾑﾘｾｯﾄ_TB
      FMOV    H0 K4B500 K6  ; ｼｰｹﾝｻ ﾊﾞｯﾃﾘ 電圧低下
      MRD
      LDP     B5F7  ; 異常追加発生
      AND     B5F6  ; 異常中
      ORP     B202  ; 干渉警報_ﾌﾞｻﾞｰ
      LD      B5F8  ; ﾌﾞｻﾞｰ出力
      ANDPI   B0F1  ; 干渉運転強行_TB
      ANDPI   B0F0  ; 干渉運転中止_TB
      ANI     B0FE  ; ﾌﾞｻﾞｰ停止_TB
      ORB
      ANB
      ANI     M7780  ; 強制出力中
      OUT     B5F8  ; ﾌﾞｻﾞｰ出力
      LDI     B202  ; 干渉警報_ﾌﾞｻﾞｰ
      LD      B202  ; 干渉警報_ﾌﾞｻﾞｰ
      AND     SM413  ; 2秒   ｸﾛｯｸ
      ORB
      ANB
      OUT     Y1019  ; 2BZ1 ﾌﾞｻﾞｰ
      MPP
      ANI     B5F6  ; 異常中
      OUT     B560  ; ｼｽﾃﾑ正常
; 
      P301
38    LD      SM52  ; ﾊﾞｯﾃﾘ低下
      OUT     B500  ; ｼｰｹﾝｻ ﾊﾞｯﾃﾘ 電圧低下
40    LD      SM0  ; 診断ｴﾗｰ
      SET     B501  ; ｼｰｹﾝｻ ｴﾗｰ
      MOV     SD0 SD50  ; 診断ｴﾗｰ番号 / ｴﾗｰ解除するｴﾗｰNO.
      AND     B0FF  ; ｱﾗｰﾑﾘｾｯﾄ_TB
      OUT     SM50  ; ｴﾗｰ解除
46    LD      T5  ; PLCRUN後_5sec
      MPS
      ANI     X59  ; TH2 油圧ﾕﾆｯﾄ油温上限
      SET     B502  ; 油温上限警報
      MRD
      ANI     X5A  ; LV1 油圧ﾕﾆｯﾄ油面下限
      SET     B503  ; 油面下限警報
      MRD
      AND     X60  ; ｵｲﾙｺﾝ　異常
      SET     B504  ; ｵｲﾙｺﾝ異常
      MRD
      ANI     X13AE  ; PH2 管端検出
      AND     M7778
      SET     B505  ; 管端検出ｾﾝｻｰｱﾗｰﾑ
      MRD
      ANI     X56  ; LS31 送り前進端
      SET     B508  ; 送り前進端
      MRD
      ANI     X57  ; LS37 送り後退限
      SET     B509  ; 送り後退端
      MPP
      AND=    K2116 D174  ; 送りMd24(807)1-1軸ﾜｰﾆﾝｸﾞ
      OUT     T272 K50  ; 送りﾊﾞｯﾃﾘ低下
      AND     T272  ; 送りﾊﾞｯﾃﾘ低下
      SET     B50A  ; 送りﾊﾞｯﾃﾘｰ電圧低下
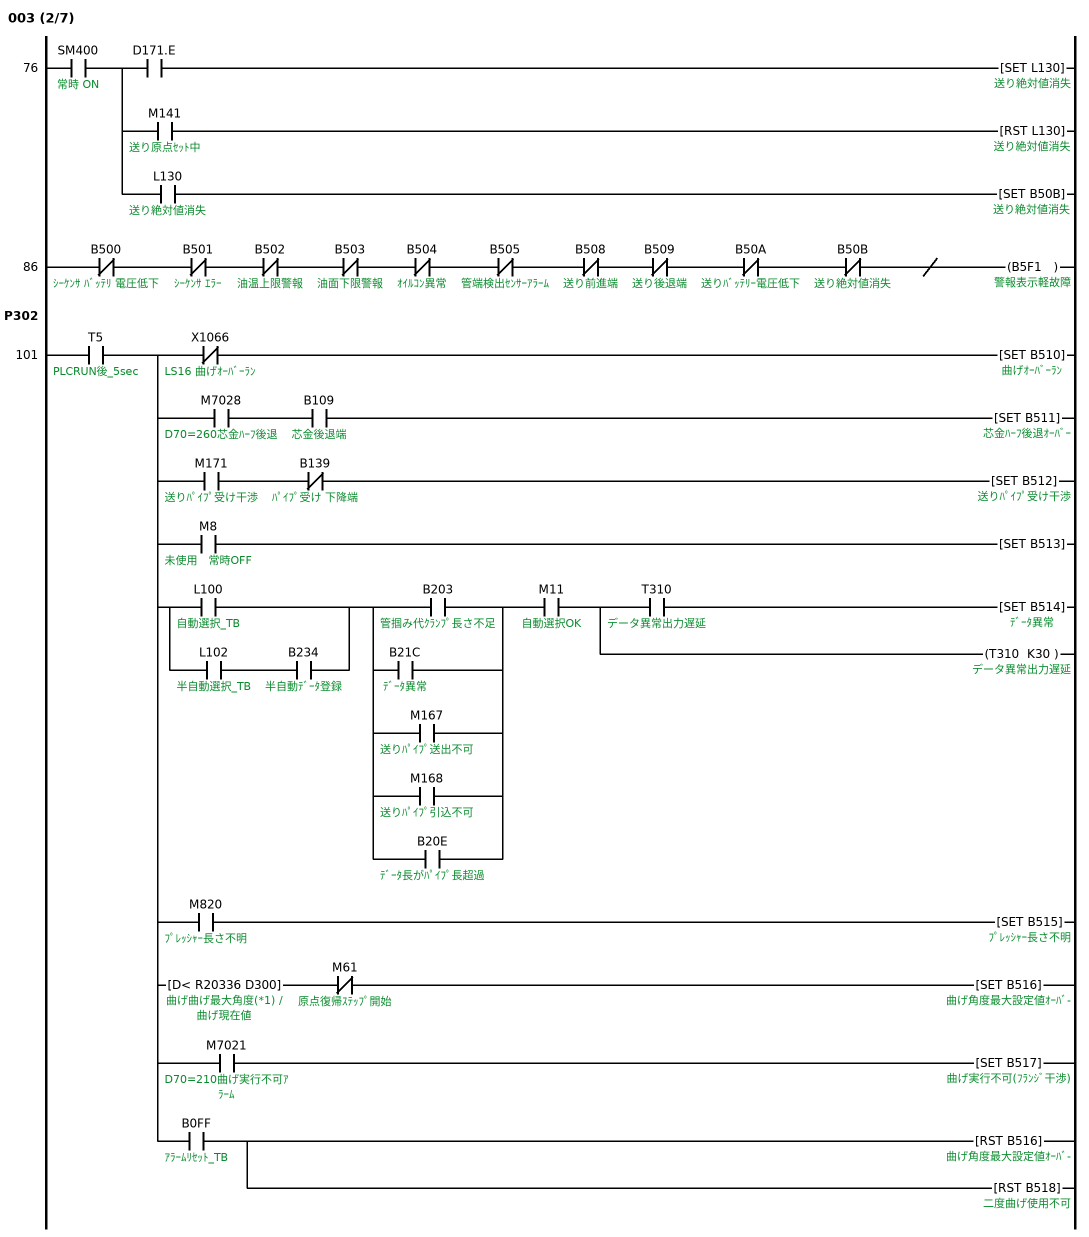
76    LD      SM400  ; 常時 ON
      MPS
      AND     D171.E
      SET     L130  ; 送り絶対値消失
      MRD
      AND     M141  ; 送り原点ｾｯﾄ中
      RST     L130  ; 送り絶対値消失
      MPP
      AND     L130  ; 送り絶対値消失
      SET     B50B  ; 送り絶対値消失
86    LDI     B500  ; ｼｰｹﾝｻ ﾊﾞｯﾃﾘ 電圧低下
      ANI     B501  ; ｼｰｹﾝｻ ｴﾗｰ
      ANI     B502  ; 油温上限警報
      ANI     B503  ; 油面下限警報
      ANI     B504  ; ｵｲﾙｺﾝ異常
      ANI     B505  ; 管端検出ｾﾝｻｰｱﾗｰﾑ
      ANI     B508  ; 送り前進端
      ANI     B509  ; 送り後退端
      ANI     B50A  ; 送りﾊﾞｯﾃﾘｰ電圧低下
      ANI     B50B  ; 送り絶対値消失
      INV
      OUT     B5F1  ; 警報表示軽故障
; 
      P302
101   LD      T5  ; PLCRUN後_5sec
      MPS
      ANI     X1066  ; LS16 曲げｵｰﾊﾞｰﾗﾝ
      SET     B510  ; 曲げｵｰﾊﾞｰﾗﾝ
      MRD
      AND     M7028  ; D70=260芯金ﾊｰﾌ後退
      AND     B109  ; 芯金後退端
      SET     B511  ; 芯金ﾊｰﾌ後退ｵｰﾊﾞｰ
      MRD
      AND     M171  ; 送りﾊﾟｲﾌﾟ受け干渉
      ANI     B139  ; ﾊﾟｲﾌﾟ受け 下降端
      SET     B512  ; 送りﾊﾟｲﾌﾟ受け干渉
      MRD
      AND     M8  ; 未使用　常時OFF
      SET     B513
      MRD
      LD      L100  ; 自動選択_TB
      LD      L102  ; 半自動選択_TB
      AND     B234  ; 半自動ﾃﾞｰﾀ登録
      ORB
      ANB
      LD      B203  ; 管掴み代ｸﾗﾝﾌﾟ長さ不足
      OR      B21C  ; ﾃﾞｰﾀ異常
      OR      M167  ; 送りﾊﾟｲﾌﾟ送出不可
      OR      M168  ; 送りﾊﾟｲﾌﾟ引込不可
      OR      B20E  ; ﾃﾞｰﾀ長がﾊﾟｲﾌﾟ長超過
      ANB
      AND     M11  ; 自動選択OK
      MPS
      AND     T310  ; データ異常出力遅延
      SET     B514  ; ﾃﾞｰﾀ異常
      MPP
      OUT     T310 K30  ; データ異常出力遅延
      MRD
      AND     M820  ; ﾌﾟﾚｯｼｬｰ長さ不明
      SET     B515  ; ﾌﾟﾚｯｼｬｰ長さ不明
      MRD
      ANDD<   R20336 D300  ; 曲げ曲げ最大角度(*1) / 曲げ現在値
      ANI     M61  ; 原点復帰ｽﾃｯﾌﾟ開始
      SET     B516  ; 曲げ角度最大設定値ｵｰﾊﾞ-
      MRD
      AND     M7021  ; D70=210曲げ実行不可ｱﾗｰﾑ
      SET     B517  ; 曲げ実行不可(ﾌﾗﾝｼﾞ干渉)
      MPP
      AND     B0FF  ; ｱﾗｰﾑﾘｾｯﾄ_TB
      RST     B516  ; 曲げ角度最大設定値ｵｰﾊﾞ-
      RST     B518  ; 二度曲げ使用不可
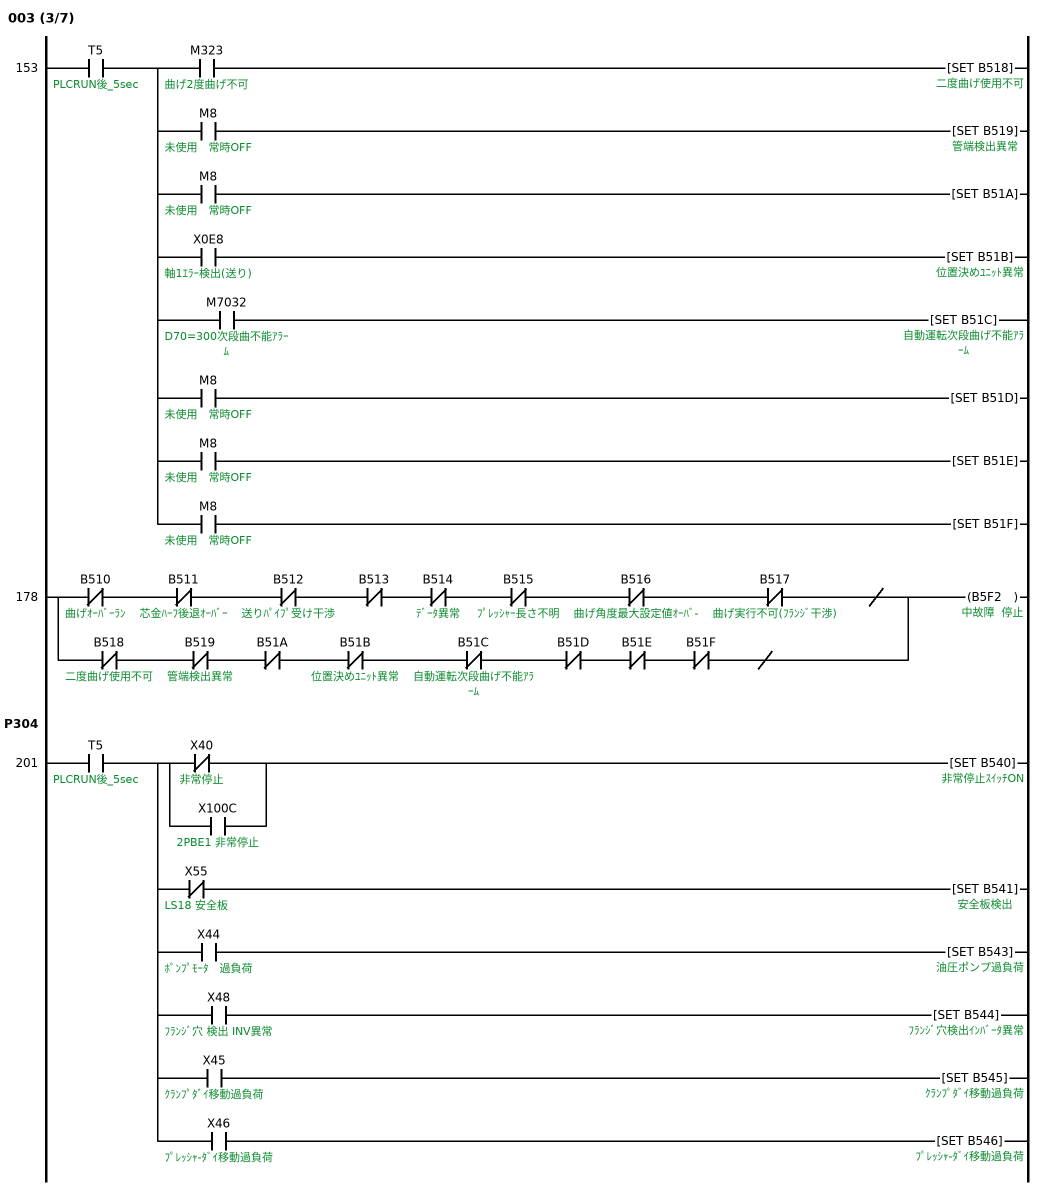
153   LD      T5  ; PLCRUN後_5sec
      MPS
      AND     M323  ; 曲げ2度曲げ不可
      SET     B518  ; 二度曲げ使用不可
      MRD
      AND     M8  ; 未使用　常時OFF
      SET     B519  ; 管端検出異常
      MRD
      AND     M8  ; 未使用　常時OFF
      SET     B51A
      MRD
      AND     X0E8  ; 軸1ｴﾗｰ検出(送り)
      SET     B51B  ; 位置決めﾕﾆｯﾄ異常
      MRD
      AND     M7032  ; D70=300次段曲不能ｱﾗｰﾑ
      SET     B51C  ; 自動運転次段曲げ不能ｱﾗｰﾑ
      MRD
      AND     M8  ; 未使用　常時OFF
      SET     B51D
      MRD
      AND     M8  ; 未使用　常時OFF
      SET     B51E
      MPP
      AND     M8  ; 未使用　常時OFF
      SET     B51F
178   LDI     B510  ; 曲げｵｰﾊﾞｰﾗﾝ
      ANI     B511  ; 芯金ﾊｰﾌ後退ｵｰﾊﾞｰ
      ANI     B512  ; 送りﾊﾟｲﾌﾟ受け干渉
      ANI     B513
      ANI     B514  ; ﾃﾞｰﾀ異常
      ANI     B515  ; ﾌﾟﾚｯｼｬｰ長さ不明
      ANI     B516  ; 曲げ角度最大設定値ｵｰﾊﾞ-
      ANI     B517  ; 曲げ実行不可(ﾌﾗﾝｼﾞ干渉)
      INV
      LDI     B518  ; 二度曲げ使用不可
      ANI     B519  ; 管端検出異常
      ANI     B51A
      ANI     B51B  ; 位置決めﾕﾆｯﾄ異常
      ANI     B51C  ; 自動運転次段曲げ不能ｱﾗｰﾑ
      ANI     B51D
      ANI     B51E
      ANI     B51F
      INV
      ORB
      OUT     B5F2  ; 中故障  停止
; 
      P304
201   LD      T5  ; PLCRUN後_5sec
      MPS
      LDI     X40  ; 非常停止
      OR      X100C  ; 2PBE1 非常停止
      ANB
      SET     B540  ; 非常停止ｽｲｯﾁON
      MRD
      ANI     X55  ; LS18 安全板
      SET     B541  ; 安全板検出
      MRD
      AND     X44  ; ﾎﾟﾝﾌﾟﾓｰﾀ　過負荷
      SET     B543  ; 油圧ポンプ過負荷
      MRD
      AND     X48  ; ﾌﾗﾝｼﾞ穴 検出 INV異常
      SET     B544  ; ﾌﾗﾝｼﾞ穴検出ｲﾝﾊﾞｰﾀ異常
      MRD
      AND     X45  ; ｸﾗﾝﾌﾟﾀﾞｲ移動過負荷
      SET     B545  ; ｸﾗﾝﾌﾟﾀﾞｲ移動過負荷
      MPP
      AND     X46  ; ﾌﾟﾚｯｼｬ-ﾀﾞｲ移動過負荷
      SET     B546  ; ﾌﾟﾚｯｼｬ-ﾀﾞｲ移動過負荷
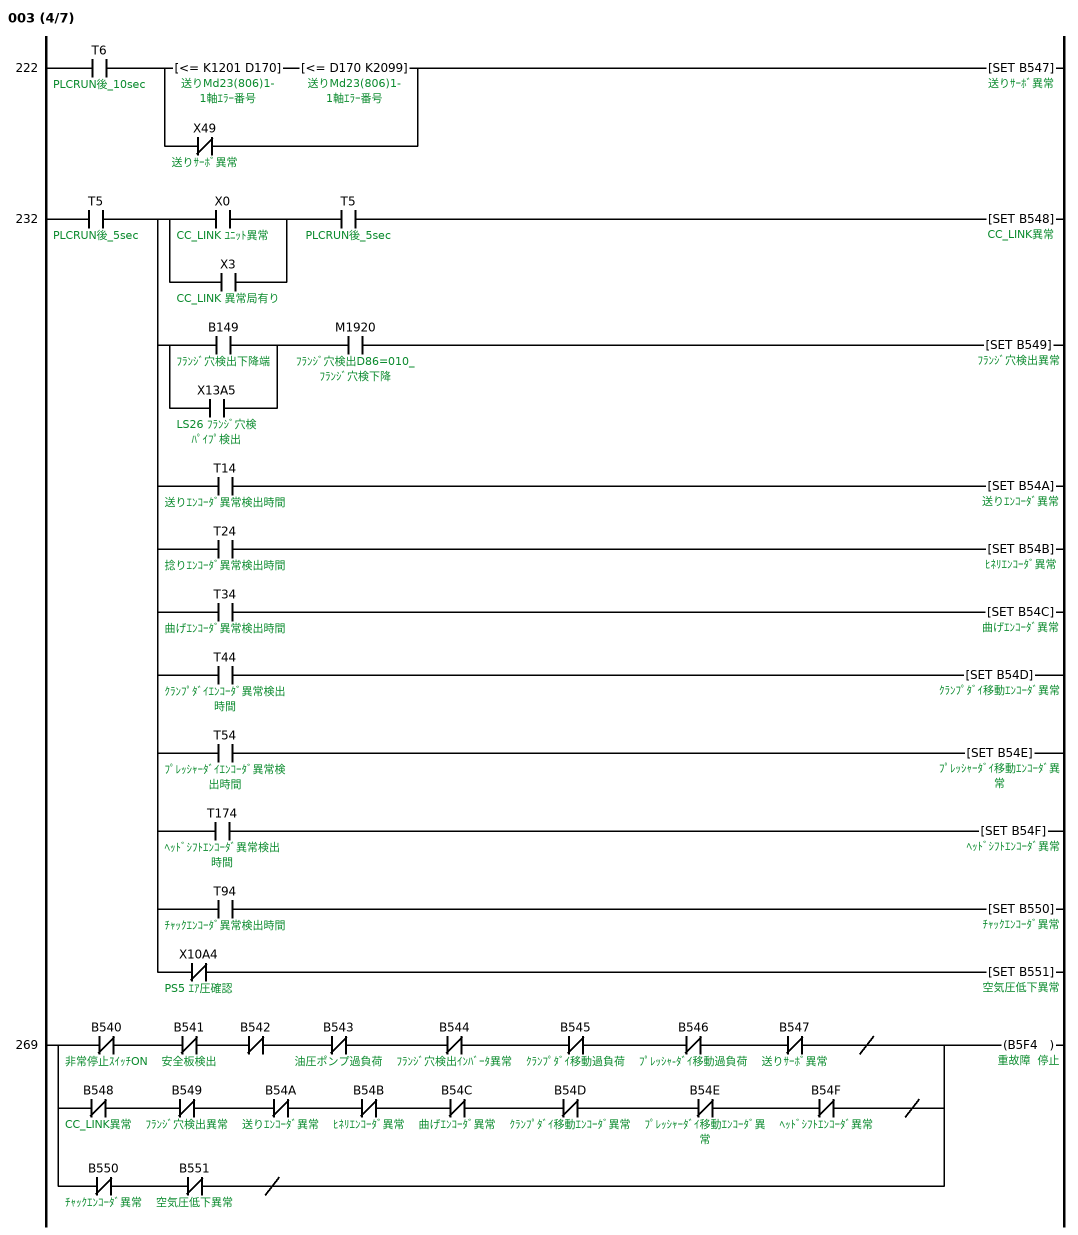
222   LD      T6  ; PLCRUN後_10sec
      LD<=    K1201 D170  ; 送りMd23(806)1-1軸ｴﾗｰ番号
      AND<=   D170 K2099  ; 送りMd23(806)1-1軸ｴﾗｰ番号
      ORI     X49  ; 送りｻｰﾎﾞ異常
      ANB
      SET     B547  ; 送りｻｰﾎﾞ異常
232   LD      T5  ; PLCRUN後_5sec
      MPS
      LD      X0  ; CC_LINK ﾕﾆｯﾄ異常
      OR      X3  ; CC_LINK 異常局有り
      ANB
      AND     T5  ; PLCRUN後_5sec
      SET     B548  ; CC_LINK異常
      MRD
      LD      B149  ; ﾌﾗﾝｼﾞ穴検出下降端
      OR      X13A5  ; LS26 ﾌﾗﾝｼﾞ穴検 ﾊﾟｲﾌﾟ検出
      ANB
      AND     M1920  ; ﾌﾗﾝｼﾞ穴検出D86=010_ﾌﾗﾝｼﾞ穴検下降
      SET     B549  ; ﾌﾗﾝｼﾞ穴検出異常
      MRD
      AND     T14  ; 送りｴﾝｺｰﾀﾞ異常検出時間
      SET     B54A  ; 送りｴﾝｺｰﾀﾞ異常
      MRD
      AND     T24  ; 捻りｴﾝｺｰﾀﾞ異常検出時間
      SET     B54B  ; ﾋﾈﾘｴﾝｺｰﾀﾞ異常
      MRD
      AND     T34  ; 曲げｴﾝｺｰﾀﾞ異常検出時間
      SET     B54C  ; 曲げｴﾝｺｰﾀﾞ異常
      MRD
      AND     T44  ; ｸﾗﾝﾌﾟﾀﾞｲｴﾝｺｰﾀﾞ異常検出時間
      SET     B54D  ; ｸﾗﾝﾌﾟﾀﾞｲ移動ｴﾝｺｰﾀﾞ異常
      MRD
      AND     T54  ; ﾌﾟﾚｯｼｬｰﾀﾞｲｴﾝｺｰﾀﾞ異常検出時間
      SET     B54E  ; ﾌﾟﾚｯｼｬｰﾀﾞｲ移動ｴﾝｺｰﾀﾞ異常
      MRD
      AND     T174  ; ﾍｯﾄﾞｼﾌﾄｴﾝｺｰﾀﾞ異常検出時間
      SET     B54F  ; ﾍｯﾄﾞｼﾌﾄｴﾝｺｰﾀﾞ異常
      MRD
      AND     T94  ; ﾁｬｯｸｴﾝｺｰﾀﾞ異常検出時間
      SET     B550  ; ﾁｬｯｸｴﾝｺｰﾀﾞ異常
      MPP
      ANI     X10A4  ; PS5 ｴｱ圧確認
      SET     B551  ; 空気圧低下異常
269   LDI     B540  ; 非常停止ｽｲｯﾁON
      ANI     B541  ; 安全板検出
      ANI     B542
      ANI     B543  ; 油圧ポンプ過負荷
      ANI     B544  ; ﾌﾗﾝｼﾞ穴検出ｲﾝﾊﾞｰﾀ異常
      ANI     B545  ; ｸﾗﾝﾌﾟﾀﾞｲ移動過負荷
      ANI     B546  ; ﾌﾟﾚｯｼｬ-ﾀﾞｲ移動過負荷
      ANI     B547  ; 送りｻｰﾎﾞ異常
      INV
      LDI     B548  ; CC_LINK異常
      ANI     B549  ; ﾌﾗﾝｼﾞ穴検出異常
      ANI     B54A  ; 送りｴﾝｺｰﾀﾞ異常
      ANI     B54B  ; ﾋﾈﾘｴﾝｺｰﾀﾞ異常
      ANI     B54C  ; 曲げｴﾝｺｰﾀﾞ異常
      ANI     B54D  ; ｸﾗﾝﾌﾟﾀﾞｲ移動ｴﾝｺｰﾀﾞ異常
      ANI     B54E  ; ﾌﾟﾚｯｼｬｰﾀﾞｲ移動ｴﾝｺｰﾀﾞ異常
      ANI     B54F  ; ﾍｯﾄﾞｼﾌﾄｴﾝｺｰﾀﾞ異常
      INV
      ORB
      LDI     B550  ; ﾁｬｯｸｴﾝｺｰﾀﾞ異常
      ANI     B551  ; 空気圧低下異常
      INV
      ORB
      OUT     B5F4  ; 重故障  停止
; 
      P305
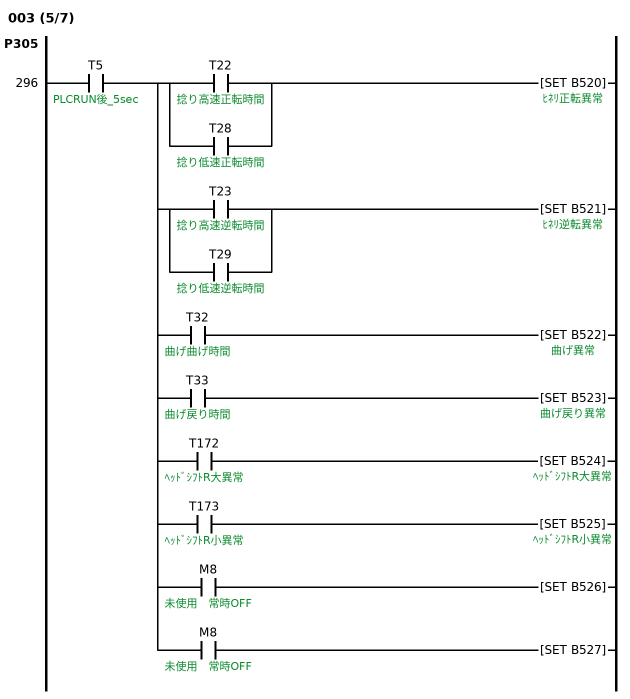
296   LD      T5  ; PLCRUN後_5sec
      MPS
      LD      T22  ; 捻り高速正転時間
      OR      T28  ; 捻り低速正転時間
      ANB
      SET     B520  ; ﾋﾈﾘ正転異常
      MRD
      LD      T23  ; 捻り高速逆転時間
      OR      T29  ; 捻り低速逆転時間
      ANB
      SET     B521  ; ﾋﾈﾘ逆転異常
      MRD
      AND     T32  ; 曲げ曲げ時間
      SET     B522  ; 曲げ異常
      MRD
      AND     T33  ; 曲げ戻り時間
      SET     B523  ; 曲げ戻り異常
      MRD
      AND     T172  ; ﾍｯﾄﾞｼﾌﾄR大異常
      SET     B524  ; ﾍｯﾄﾞｼﾌﾄR大異常
      MRD
      AND     T173  ; ﾍｯﾄﾞｼﾌﾄR小異常
      SET     B525  ; ﾍｯﾄﾞｼﾌﾄR小異常
      MRD
      AND     M8  ; 未使用　常時OFF
      SET     B526
      MPP
      AND     M8  ; 未使用　常時OFF
      SET     B527
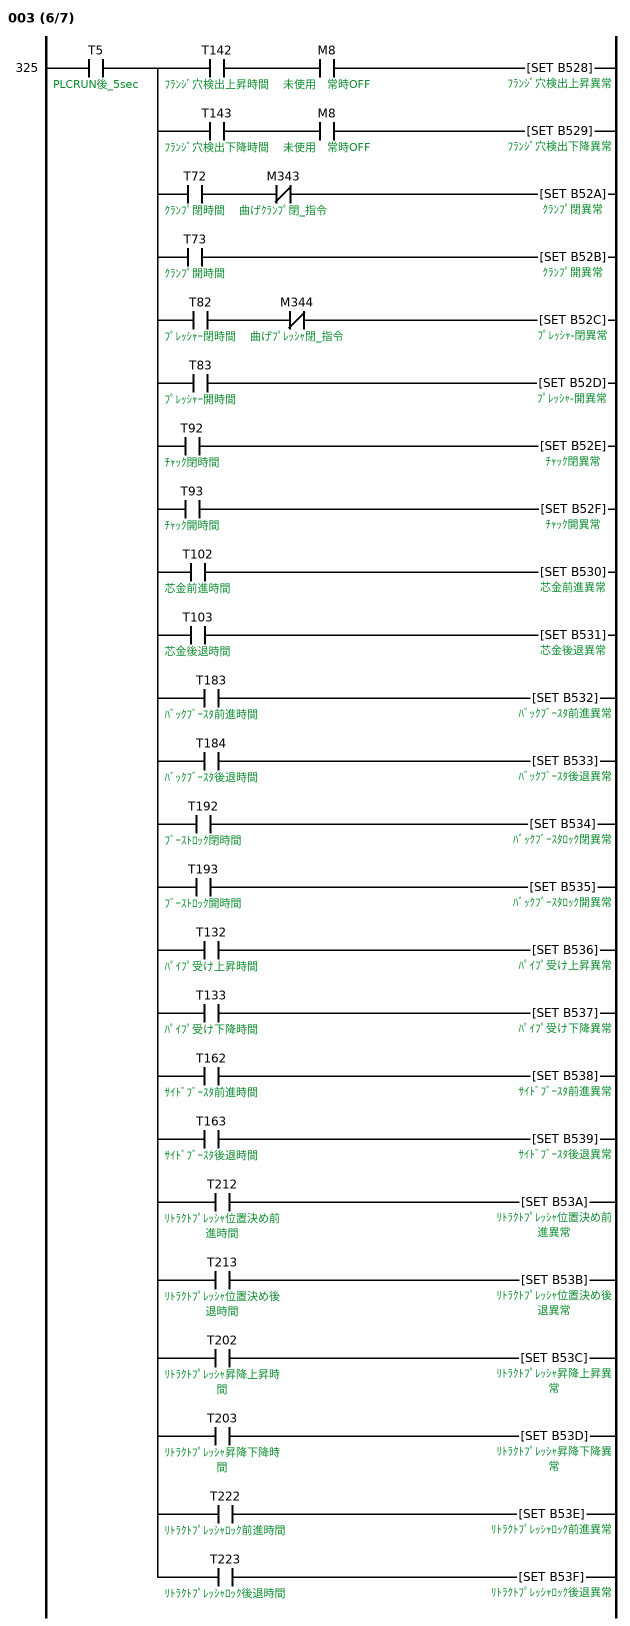
325   LD      T5  ; PLCRUN後_5sec
      MPS
      AND     T142  ; ﾌﾗﾝｼﾞ穴検出上昇時間
      AND     M8  ; 未使用　常時OFF
      SET     B528  ; ﾌﾗﾝｼﾞ穴検出上昇異常
      MRD
      AND     T143  ; ﾌﾗﾝｼﾞ穴検出下降時間
      AND     M8  ; 未使用　常時OFF
      SET     B529  ; ﾌﾗﾝｼﾞ穴検出下降異常
      MRD
      AND     T72  ; ｸﾗﾝﾌﾟ閉時間
      ANI     M343  ; 曲げｸﾗﾝﾌﾟ閉_指令
      SET     B52A  ; ｸﾗﾝﾌﾟ閉異常
      MRD
      AND     T73  ; ｸﾗﾝﾌﾟ開時間
      SET     B52B  ; ｸﾗﾝﾌﾟ開異常
      MRD
      AND     T82  ; ﾌﾟﾚｯｼｬｰ閉時間
      ANI     M344  ; 曲げﾌﾟﾚｯｼｬ閉_指令
      SET     B52C  ; ﾌﾟﾚｯｼｬ-閉異常
      MRD
      AND     T83  ; ﾌﾟﾚｯｼｬｰ開時間
      SET     B52D  ; ﾌﾟﾚｯｼｬ-開異常
      MRD
      AND     T92  ; ﾁｬｯｸ閉時間
      SET     B52E  ; ﾁｬｯｸ閉異常
      MRD
      AND     T93  ; ﾁｬｯｸ開時間
      SET     B52F  ; ﾁｬｯｸ開異常
      MRD
      AND     T102  ; 芯金前進時間
      SET     B530  ; 芯金前進異常
      MRD
      AND     T103  ; 芯金後退時間
      SET     B531  ; 芯金後退異常
      MRD
      AND     T183  ; ﾊﾞｯｸﾌﾞｰｽﾀ前進時間
      SET     B532  ; ﾊﾞｯｸﾌﾞｰｽﾀ前進異常
      MRD
      AND     T184  ; ﾊﾞｯｸﾌﾞｰｽﾀ後退時間
      SET     B533  ; ﾊﾞｯｸﾌﾞｰｽﾀ後退異常
      MRD
      AND     T192  ; ﾌﾞｰｽﾄﾛｯｸ閉時間
      SET     B534  ; ﾊﾞｯｸﾌﾞｰｽﾀﾛｯｸ閉異常
      MRD
      AND     T193  ; ﾌﾞｰｽﾄﾛｯｸ開時間
      SET     B535  ; ﾊﾞｯｸﾌﾞｰｽﾀﾛｯｸ開異常
      MRD
      AND     T132  ; ﾊﾟｲﾌﾟ受け上昇時間
      SET     B536  ; ﾊﾟｲﾌﾟ受け上昇異常
      MRD
      AND     T133  ; ﾊﾟｲﾌﾟ受け下降時間
      SET     B537  ; ﾊﾟｲﾌﾟ受け下降異常
      MRD
      AND     T162  ; ｻｲﾄﾞﾌﾞｰｽﾀ前進時間
      SET     B538  ; ｻｲﾄﾞﾌﾞｰｽﾀ前進異常
      MRD
      AND     T163  ; ｻｲﾄﾞﾌﾞｰｽﾀ後退時間
      SET     B539  ; ｻｲﾄﾞﾌﾞｰｽﾀ後退異常
      MRD
      AND     T212  ; ﾘﾄﾗｸﾄﾌﾟﾚｯｼｬ位置決め前進時間
      SET     B53A  ; ﾘﾄﾗｸﾄﾌﾟﾚｯｼｬ位置決め前進異常
      MRD
      AND     T213  ; ﾘﾄﾗｸﾄﾌﾟﾚｯｼｬ位置決め後退時間
      SET     B53B  ; ﾘﾄﾗｸﾄﾌﾟﾚｯｼｬ位置決め後退異常
      MRD
      AND     T202  ; ﾘﾄﾗｸﾄﾌﾟﾚｯｼｬ昇降上昇時間
      SET     B53C  ; ﾘﾄﾗｸﾄﾌﾟﾚｯｼｬ昇降上昇異常
      MRD
      AND     T203  ; ﾘﾄﾗｸﾄﾌﾟﾚｯｼｬ昇降下降時間
      SET     B53D  ; ﾘﾄﾗｸﾄﾌﾟﾚｯｼｬ昇降下降異常
      MRD
      AND     T222  ; ﾘﾄﾗｸﾄﾌﾟﾚｯｼｬﾛｯｸ前進時間
      SET     B53E  ; ﾘﾄﾗｸﾄﾌﾟﾚｯｼｬﾛｯｸ前進異常
      MPP
      AND     T223  ; ﾘﾄﾗｸﾄﾌﾟﾚｯｼｬﾛｯｸ後退時間
      SET     B53F  ; ﾘﾄﾗｸﾄﾌﾟﾚｯｼｬﾛｯｸ後退異常
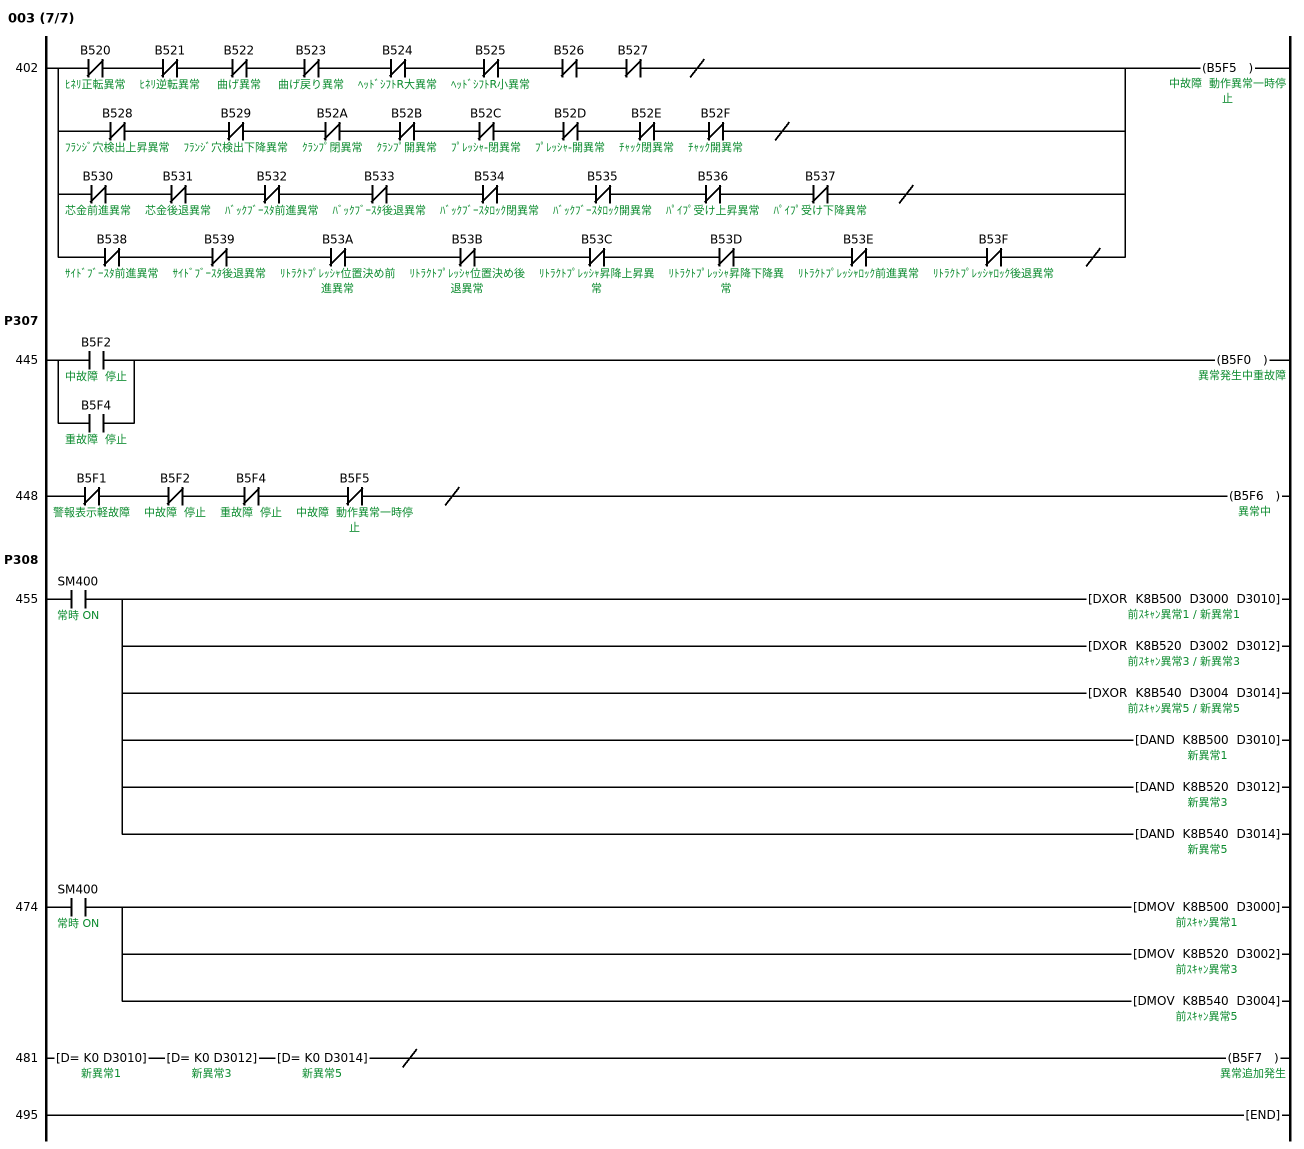
402   LDI     B520  ; ﾋﾈﾘ正転異常
      ANI     B521  ; ﾋﾈﾘ逆転異常
      ANI     B522  ; 曲げ異常
      ANI     B523  ; 曲げ戻り異常
      ANI     B524  ; ﾍｯﾄﾞｼﾌﾄR大異常
      ANI     B525  ; ﾍｯﾄﾞｼﾌﾄR小異常
      ANI     B526
      ANI     B527
      INV
      LDI     B528  ; ﾌﾗﾝｼﾞ穴検出上昇異常
      ANI     B529  ; ﾌﾗﾝｼﾞ穴検出下降異常
      ANI     B52A  ; ｸﾗﾝﾌﾟ閉異常
      ANI     B52B  ; ｸﾗﾝﾌﾟ開異常
      ANI     B52C  ; ﾌﾟﾚｯｼｬ-閉異常
      ANI     B52D  ; ﾌﾟﾚｯｼｬ-開異常
      ANI     B52E  ; ﾁｬｯｸ閉異常
      ANI     B52F  ; ﾁｬｯｸ開異常
      INV
      ORB
      LDI     B530  ; 芯金前進異常
      ANI     B531  ; 芯金後退異常
      ANI     B532  ; ﾊﾞｯｸﾌﾞｰｽﾀ前進異常
      ANI     B533  ; ﾊﾞｯｸﾌﾞｰｽﾀ後退異常
      ANI     B534  ; ﾊﾞｯｸﾌﾞｰｽﾀﾛｯｸ閉異常
      ANI     B535  ; ﾊﾞｯｸﾌﾞｰｽﾀﾛｯｸ開異常
      ANI     B536  ; ﾊﾟｲﾌﾟ受け上昇異常
      ANI     B537  ; ﾊﾟｲﾌﾟ受け下降異常
      INV
      ORB
      LDI     B538  ; ｻｲﾄﾞﾌﾞｰｽﾀ前進異常
      ANI     B539  ; ｻｲﾄﾞﾌﾞｰｽﾀ後退異常
      ANI     B53A  ; ﾘﾄﾗｸﾄﾌﾟﾚｯｼｬ位置決め前進異常
      ANI     B53B  ; ﾘﾄﾗｸﾄﾌﾟﾚｯｼｬ位置決め後退異常
      ANI     B53C  ; ﾘﾄﾗｸﾄﾌﾟﾚｯｼｬ昇降上昇異常
      ANI     B53D  ; ﾘﾄﾗｸﾄﾌﾟﾚｯｼｬ昇降下降異常
      ANI     B53E  ; ﾘﾄﾗｸﾄﾌﾟﾚｯｼｬﾛｯｸ前進異常
      ANI     B53F  ; ﾘﾄﾗｸﾄﾌﾟﾚｯｼｬﾛｯｸ後退異常
      INV
      ORB
      OUT     B5F5  ; 中故障  動作異常一時停止
; 
      P307
445   LD      B5F2  ; 中故障  停止
      OR      B5F4  ; 重故障  停止
      OUT     B5F0  ; 異常発生中重故障
448   LDI     B5F1  ; 警報表示軽故障
      ANI     B5F2  ; 中故障  停止
      ANI     B5F4  ; 重故障  停止
      ANI     B5F5  ; 中故障  動作異常一時停止
      INV
      OUT     B5F6  ; 異常中
      P308
455   LD      SM400  ; 常時 ON
      DXOR    K8B500 D3000 D3010  ; 前ｽｷｬﾝ異常1 / 新異常1
      DXOR    K8B520 D3002 D3012  ; 前ｽｷｬﾝ異常3 / 新異常3
      DXOR    K8B540 D3004 D3014  ; 前ｽｷｬﾝ異常5 / 新異常5
      DAND    K8B500 D3010
      DAND    K8B520 D3012
      DAND    K8B540 D3014
474   LD      SM400  ; 常時 ON
      DMOV    K8B500 D3000
      DMOV    K8B520 D3002
      DMOV    K8B540 D3004
481   LDD=    K0 D3010  ; 新異常1
      ANDD=   K0 D3012  ; 新異常3
      ANDD=   K0 D3014  ; 新異常5
      INV
      OUT     B5F7  ; 異常追加発生
495   END
END_PROGRAM

PROGRAM 004  // 運転準備
      P400
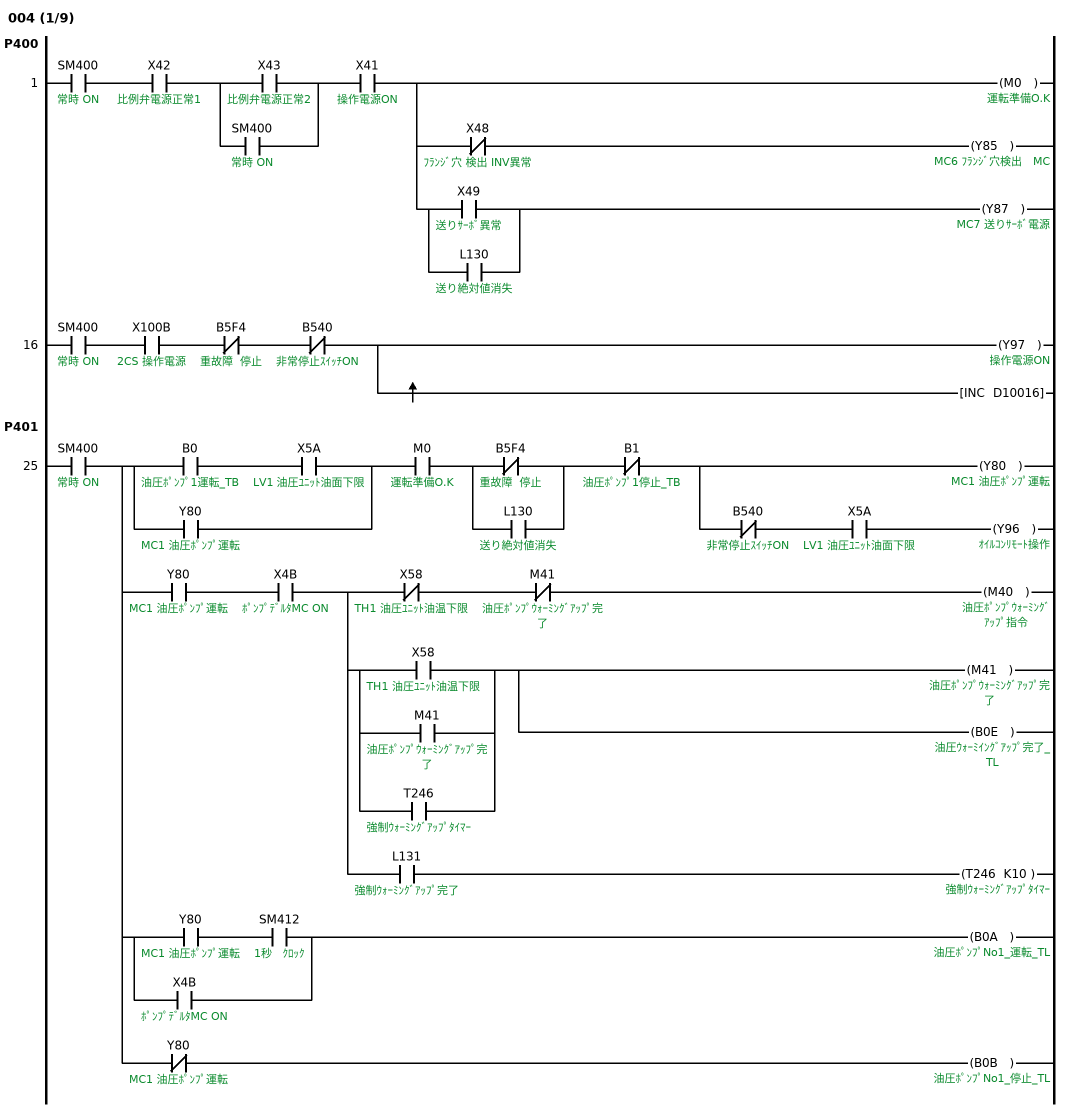
1     LD      SM400  ; 常時 ON
      AND     X42  ; 比例弁電源正常1
      LD      X43  ; 比例弁電源正常2
      OR      SM400  ; 常時 ON
      ANB
      AND     X41  ; 操作電源ON
      OUT     M0  ; 運転準備O.K
      MPS
      ANI     X48  ; ﾌﾗﾝｼﾞ穴 検出 INV異常
      OUT     Y85  ; MC6 ﾌﾗﾝｼﾞ穴検出　MC
      MPP
      LD      X49  ; 送りｻｰﾎﾞ異常
      OR      L130  ; 送り絶対値消失
      ANB
      OUT     Y87  ; MC7 送りｻｰﾎﾞ電源
16    LD      SM400  ; 常時 ON
      AND     X100B  ; 2CS 操作電源
      ANI     B5F4  ; 重故障  停止
      ANI     B540  ; 非常停止ｽｲｯﾁON
      OUT     Y97  ; 操作電源ON
      MEP
      INC     D10016
      P401
25    LD      SM400  ; 常時 ON
      MPS
      LD      B0  ; 油圧ﾎﾟﾝﾌﾟ1運転_TB
      AND     X5A  ; LV1 油圧ﾕﾆｯﾄ油面下限
      OR      Y80  ; MC1 油圧ﾎﾟﾝﾌﾟ運転
      ANB
      AND     M0  ; 運転準備O.K
      LDI     B5F4  ; 重故障  停止
      OR      L130  ; 送り絶対値消失
      ANB
      ANI     B1  ; 油圧ﾎﾟﾝﾌﾟ1停止_TB
      OUT     Y80  ; MC1 油圧ﾎﾟﾝﾌﾟ運転
      ANI     B540  ; 非常停止ｽｲｯﾁON
      AND     X5A  ; LV1 油圧ﾕﾆｯﾄ油面下限
      OUT     Y96  ; ｵｲﾙｺﾝﾘﾓｰﾄ操作
      MRD
      AND     Y80  ; MC1 油圧ﾎﾟﾝﾌﾟ運転
      AND     X4B  ; ﾎﾟﾝﾌﾟﾃﾞﾙﾀMC ON
      MPS
      ANI     X58  ; TH1 油圧ﾕﾆｯﾄ油温下限
      ANI     M41  ; 油圧ﾎﾟﾝﾌﾟｳｫｰﾐﾝｸﾞｱｯﾌﾟ完了
      OUT     M40  ; 油圧ﾎﾟﾝﾌﾟｳｫｰﾐﾝｸﾞ ｱｯﾌﾟ指令
      MRD
      LD      X58  ; TH1 油圧ﾕﾆｯﾄ油温下限
      OR      M41  ; 油圧ﾎﾟﾝﾌﾟｳｫｰﾐﾝｸﾞｱｯﾌﾟ完了
      OR      T246  ; 強制ｳｫｰﾐﾝｸﾞｱｯﾌﾟﾀｲﾏｰ
      ANB
      OUT     M41  ; 油圧ﾎﾟﾝﾌﾟｳｫｰﾐﾝｸﾞｱｯﾌﾟ完了
      OUT     B0E  ; 油圧ｳｫｰﾐｲﾝｸﾞｱｯﾌﾟ完了_TL
      MPP
      AND     L131  ; 強制ｳｫｰﾐﾝｸﾞｱｯﾌﾟ完了
      OUT     T246 K10  ; 強制ｳｫｰﾐﾝｸﾞｱｯﾌﾟﾀｲﾏｰ
      MRD
      LD      Y80  ; MC1 油圧ﾎﾟﾝﾌﾟ運転
      AND     SM412  ; 1秒   ｸﾛｯｸ
      OR      X4B  ; ﾎﾟﾝﾌﾟﾃﾞﾙﾀMC ON
      ANB
      OUT     B0A  ; 油圧ﾎﾟﾝﾌﾟNo1_運転_TL
      MPP
      ANI     Y80  ; MC1 油圧ﾎﾟﾝﾌﾟ運転
      OUT     B0B  ; 油圧ﾎﾟﾝﾌﾟNo1_停止_TL
; 
      P402
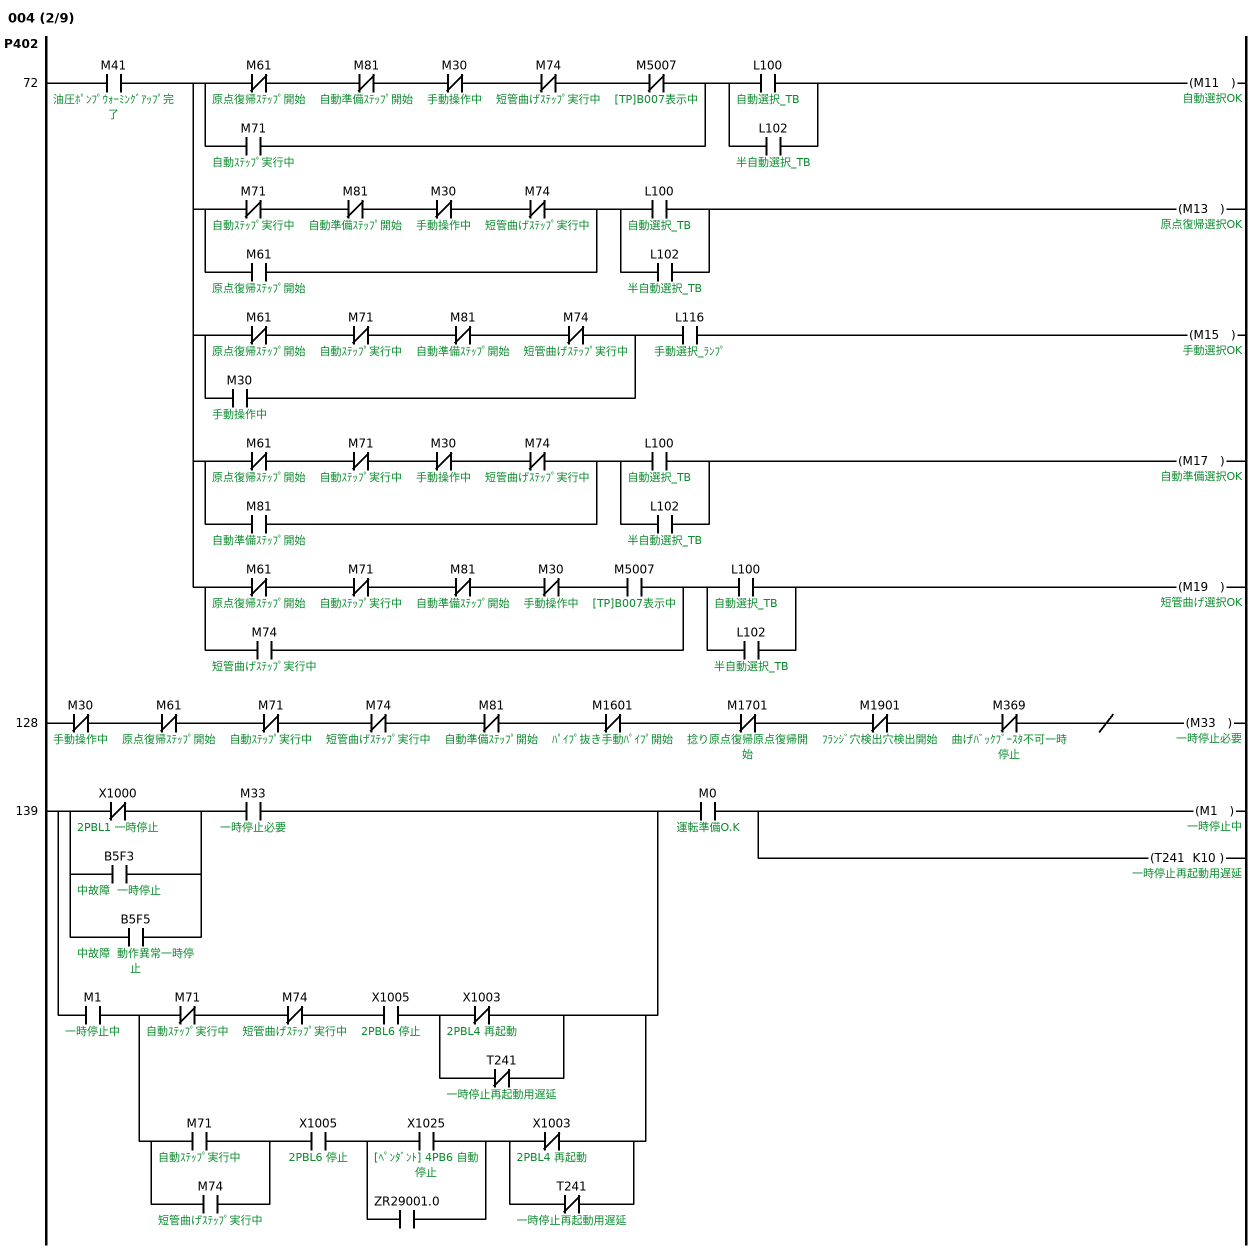
72    LD      M41  ; 油圧ﾎﾟﾝﾌﾟｳｫｰﾐﾝｸﾞｱｯﾌﾟ完了
      MPS
      LDI     M61  ; 原点復帰ｽﾃｯﾌﾟ開始
      ANI     M81  ; 自動準備ｽﾃｯﾌﾟ開始
      ANI     M30  ; 手動操作中
      ANI     M74  ; 短管曲げｽﾃｯﾌﾟ実行中
      ANI     M5007  ; [TP]B007表示中
      OR      M71  ; 自動ｽﾃｯﾌﾟ実行中
      ANB
      LD      L100  ; 自動選択_TB
      OR      L102  ; 半自動選択_TB
      ANB
      OUT     M11  ; 自動選択OK
      MRD
      LDI     M71  ; 自動ｽﾃｯﾌﾟ実行中
      ANI     M81  ; 自動準備ｽﾃｯﾌﾟ開始
      ANI     M30  ; 手動操作中
      ANI     M74  ; 短管曲げｽﾃｯﾌﾟ実行中
      OR      M61  ; 原点復帰ｽﾃｯﾌﾟ開始
      ANB
      LD      L100  ; 自動選択_TB
      OR      L102  ; 半自動選択_TB
      ANB
      OUT     M13  ; 原点復帰選択OK
      MRD
      LDI     M61  ; 原点復帰ｽﾃｯﾌﾟ開始
      ANI     M71  ; 自動ｽﾃｯﾌﾟ実行中
      ANI     M81  ; 自動準備ｽﾃｯﾌﾟ開始
      ANI     M74  ; 短管曲げｽﾃｯﾌﾟ実行中
      OR      M30  ; 手動操作中
      ANB
      AND     L116  ; 手動選択_ﾗﾝﾌﾟ
      OUT     M15  ; 手動選択OK
      MRD
      LDI     M61  ; 原点復帰ｽﾃｯﾌﾟ開始
      ANI     M71  ; 自動ｽﾃｯﾌﾟ実行中
      ANI     M30  ; 手動操作中
      ANI     M74  ; 短管曲げｽﾃｯﾌﾟ実行中
      OR      M81  ; 自動準備ｽﾃｯﾌﾟ開始
      ANB
      LD      L100  ; 自動選択_TB
      OR      L102  ; 半自動選択_TB
      ANB
      OUT     M17  ; 自動準備選択OK
      MPP
      LDI     M61  ; 原点復帰ｽﾃｯﾌﾟ開始
      ANI     M71  ; 自動ｽﾃｯﾌﾟ実行中
      ANI     M81  ; 自動準備ｽﾃｯﾌﾟ開始
      ANI     M30  ; 手動操作中
      AND     M5007  ; [TP]B007表示中
      OR      M74  ; 短管曲げｽﾃｯﾌﾟ実行中
      ANB
      LD      L100  ; 自動選択_TB
      OR      L102  ; 半自動選択_TB
      ANB
      OUT     M19  ; 短管曲げ選択OK
128   LDI     M30  ; 手動操作中
      ANI     M61  ; 原点復帰ｽﾃｯﾌﾟ開始
      ANI     M71  ; 自動ｽﾃｯﾌﾟ実行中
      ANI     M74  ; 短管曲げｽﾃｯﾌﾟ実行中
      ANI     M81  ; 自動準備ｽﾃｯﾌﾟ開始
      ANI     M1601  ; ﾊﾟｲﾌﾟ抜き手動ﾊﾟｲﾌﾟ開始
      ANI     M1701  ; 捻り原点復帰原点復帰開始
      ANI     M1901  ; ﾌﾗﾝｼﾞ穴検出穴検出開始
      ANI     M369  ; 曲げﾊﾞｯｸﾌﾞｰｽﾀ不可一時停止
      INV
      OUT     M33  ; 一時停止必要
139   LDI     X1000  ; 2PBL1 一時停止
      OR      B5F3  ; 中故障  一時停止
      OR      B5F5  ; 中故障  動作異常一時停止
      AND     M33  ; 一時停止必要
      LD      M1  ; 一時停止中
      LDI     M71  ; 自動ｽﾃｯﾌﾟ実行中
      ANI     M74  ; 短管曲げｽﾃｯﾌﾟ実行中
      AND     X1005  ; 2PBL6 停止
      LDI     X1003  ; 2PBL4 再起動
      ORI     T241  ; 一時停止再起動用遅延
      ANB
      LD      M71  ; 自動ｽﾃｯﾌﾟ実行中
      OR      M74  ; 短管曲げｽﾃｯﾌﾟ実行中
      AND     X1005  ; 2PBL6 停止
      LD      X1025  ; [ﾍﾟﾝﾀﾞﾝﾄ] 4PB6 自動 停止
      OR      ZR29001.0
      ANB
      LDI     X1003  ; 2PBL4 再起動
      ORI     T241  ; 一時停止再起動用遅延
      ANB
      ORB
      ANB
      ORB
      AND     M0  ; 運転準備O.K
      OUT     M1  ; 一時停止中
      OUT     T241 K10  ; 一時停止再起動用遅延
      P413
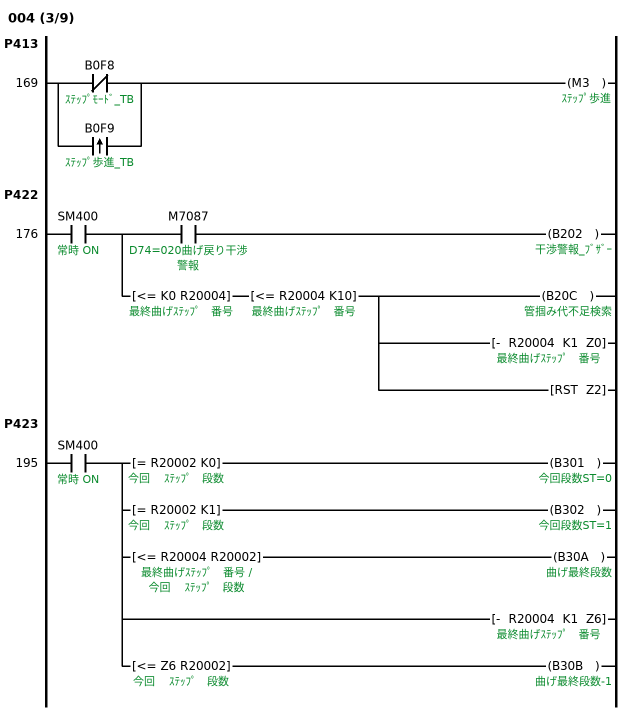
169   LDI     B0F8  ; ｽﾃｯﾌﾟﾓｰﾄﾞ_TB
      ORP     B0F9  ; ｽﾃｯﾌﾟ歩進_TB
      OUT     M3  ; ｽﾃｯﾌﾟ歩進
; 
      P422
176   LD      SM400  ; 常時 ON
      MPS
      AND     M7087  ; D74=020曲げ戻り干渉警報
      OUT     B202  ; 干渉警報_ﾌﾞｻﾞｰ
      MPP
      AND<=   K0 R20004  ; 最終曲げｽﾃｯﾌﾟ   番号
      AND<=   R20004 K10  ; 最終曲げｽﾃｯﾌﾟ   番号
      OUT     B20C  ; 管掴み代不足検索
      -       R20004 K1 Z0
      RST     Z2
; 
      P423
195   LD      SM400  ; 常時 ON
      MPS
      AND=    R20002 K0  ; 今回    ｽﾃｯﾌﾟ   段数
      OUT     B301  ; 今回段数ST=0
      MRD
      AND=    R20002 K1  ; 今回    ｽﾃｯﾌﾟ   段数
      OUT     B302  ; 今回段数ST=1
      MRD
      AND<=   R20004 R20002  ; 最終曲げｽﾃｯﾌﾟ   番号 / 今回    ｽﾃｯﾌﾟ   段数
      OUT     B30A  ; 曲げ最終段数
      MPP
      -       R20004 K1 Z6
      AND<=   Z6 R20002  ; 今回    ｽﾃｯﾌﾟ   段数
      OUT     B30B  ; 曲げ最終段数-1
; 
      P424
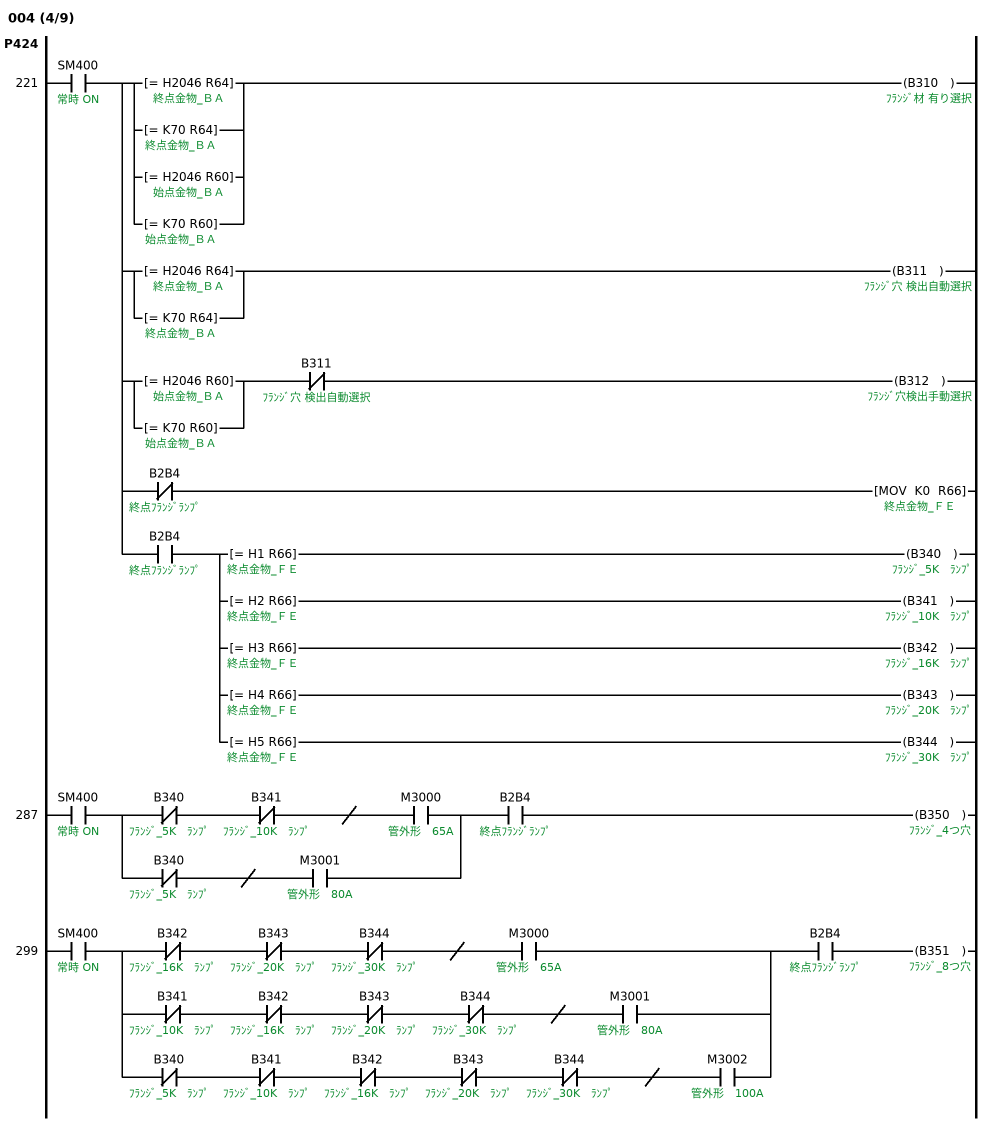
221   LD      SM400  ; 常時 ON
      MPS
      LD=     H2046 R64  ; 終点金物_ＢＡ
      OR=     K70 R64  ; 終点金物_ＢＡ
      OR=     H2046 R60  ; 始点金物_ＢＡ
      OR=     K70 R60  ; 始点金物_ＢＡ
      ANB
      OUT     B310  ; ﾌﾗﾝｼﾞ材 有り選択
      MRD
      LD=     H2046 R64  ; 終点金物_ＢＡ
      OR=     K70 R64  ; 終点金物_ＢＡ
      ANB
      OUT     B311  ; ﾌﾗﾝｼﾞ穴 検出自動選択
      MRD
      LD=     H2046 R60  ; 始点金物_ＢＡ
      OR=     K70 R60  ; 始点金物_ＢＡ
      ANB
      ANI     B311  ; ﾌﾗﾝｼﾞ穴 検出自動選択
      OUT     B312  ; ﾌﾗﾝｼﾞ穴検出手動選択
      MRD
      ANI     B2B4  ; 終点ﾌﾗﾝｼﾞﾗﾝﾌﾟ
      MOV     K0 R66  ; 終点金物_ＦＥ
      MPP
      AND     B2B4  ; 終点ﾌﾗﾝｼﾞﾗﾝﾌﾟ
      MPS
      AND=    H1 R66  ; 終点金物_ＦＥ
      OUT     B340  ; ﾌﾗﾝｼﾞ_5K　ﾗﾝﾌﾟ
      MRD
      AND=    H2 R66  ; 終点金物_ＦＥ
      OUT     B341  ; ﾌﾗﾝｼﾞ_10K　ﾗﾝﾌﾟ
      MRD
      AND=    H3 R66  ; 終点金物_ＦＥ
      OUT     B342  ; ﾌﾗﾝｼﾞ_16K　ﾗﾝﾌﾟ
      MRD
      AND=    H4 R66  ; 終点金物_ＦＥ
      OUT     B343  ; ﾌﾗﾝｼﾞ_20K　ﾗﾝﾌﾟ
      MPP
      AND=    H5 R66  ; 終点金物_ＦＥ
      OUT     B344  ; ﾌﾗﾝｼﾞ_30K　ﾗﾝﾌﾟ
287   LD      SM400  ; 常時 ON
      LDI     B340  ; ﾌﾗﾝｼﾞ_5K　ﾗﾝﾌﾟ
      ANI     B341  ; ﾌﾗﾝｼﾞ_10K　ﾗﾝﾌﾟ
      INV
      AND     M3000  ; 管外形　65A
      LDI     B340  ; ﾌﾗﾝｼﾞ_5K　ﾗﾝﾌﾟ
      INV
      AND     M3001  ; 管外形　80A
      ORB
      ANB
      AND     B2B4  ; 終点ﾌﾗﾝｼﾞﾗﾝﾌﾟ
      OUT     B350  ; ﾌﾗﾝｼﾞ_4つ穴
299   LD      SM400  ; 常時 ON
      LDI     B342  ; ﾌﾗﾝｼﾞ_16K　ﾗﾝﾌﾟ
      ANI     B343  ; ﾌﾗﾝｼﾞ_20K　ﾗﾝﾌﾟ
      ANI     B344  ; ﾌﾗﾝｼﾞ_30K　ﾗﾝﾌﾟ
      INV
      AND     M3000  ; 管外形　65A
      LDI     B341  ; ﾌﾗﾝｼﾞ_10K　ﾗﾝﾌﾟ
      ANI     B342  ; ﾌﾗﾝｼﾞ_16K　ﾗﾝﾌﾟ
      ANI     B343  ; ﾌﾗﾝｼﾞ_20K　ﾗﾝﾌﾟ
      ANI     B344  ; ﾌﾗﾝｼﾞ_30K　ﾗﾝﾌﾟ
      INV
      AND     M3001  ; 管外形　80A
      ORB
      LDI     B340  ; ﾌﾗﾝｼﾞ_5K　ﾗﾝﾌﾟ
      ANI     B341  ; ﾌﾗﾝｼﾞ_10K　ﾗﾝﾌﾟ
      ANI     B342  ; ﾌﾗﾝｼﾞ_16K　ﾗﾝﾌﾟ
      ANI     B343  ; ﾌﾗﾝｼﾞ_20K　ﾗﾝﾌﾟ
      ANI     B344  ; ﾌﾗﾝｼﾞ_30K　ﾗﾝﾌﾟ
      INV
      AND     M3002  ; 管外形　100A
      ORB
      ANB
      AND     B2B4  ; 終点ﾌﾗﾝｼﾞﾗﾝﾌﾟ
      OUT     B351  ; ﾌﾗﾝｼﾞ_8つ穴
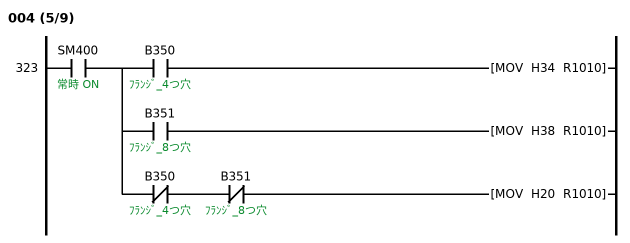
323   LD      SM400  ; 常時 ON
      MPS
      AND     B350  ; ﾌﾗﾝｼﾞ_4つ穴
      MOV     H34 R1010
      MRD
      AND     B351  ; ﾌﾗﾝｼﾞ_8つ穴
      MOV     H38 R1010
      MPP
      ANI     B350  ; ﾌﾗﾝｼﾞ_4つ穴
      ANI     B351  ; ﾌﾗﾝｼﾞ_8つ穴
      MOV     H20 R1010
; 
      P430
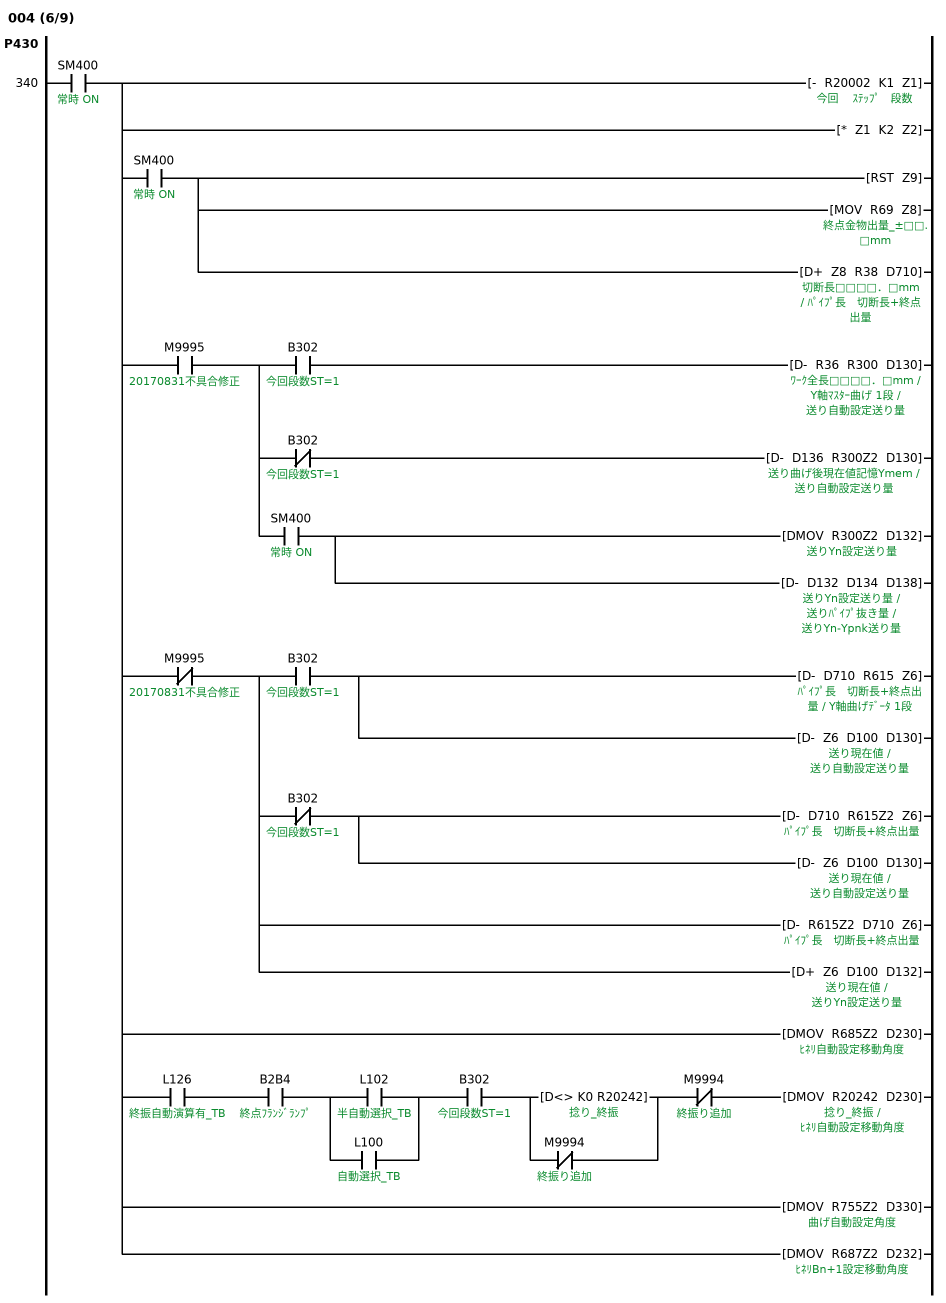
340   LD      SM400  ; 常時 ON
      -       R20002 K1 Z1
      *       Z1 K2 Z2
      MPS
      AND     SM400  ; 常時 ON
      RST     Z9
      MOV     R69 Z8  ; 終点金物出量_±□□.□mm
      D+      Z8 R38 D710  ; 切断長□□□□．□mm / ﾊﾟｲﾌﾟ長　切断長+終点出量
      MRD
      AND     M9995  ; 20170831不具合修正
      MPS
      AND     B302  ; 今回段数ST=1
      D-      R36 R300 D130  ; ﾜｰｸ全長□□□□．□mm / Y軸ﾏｽﾀｰ曲げ 1段 / 送り自動設定送り量
      MRD
      ANI     B302  ; 今回段数ST=1
      D-      D136 R300Z2 D130  ; 送り曲げ後現在値記憶Ymem
      MPP
      AND     SM400  ; 常時 ON
      DMOV    R300Z2 D132  ; 送りYn設定送り量
      D-      D132 D134 D138  ; 送りﾊﾟｲﾌﾟ抜き量 / 送りYn-Ypnk送り量
      MRD
      ANI     M9995  ; 20170831不具合修正
      MPS
      AND     B302  ; 今回段数ST=1
      D-      D710 R615 Z6  ; Y軸曲げﾃﾞｰﾀ 1段
      D-      Z6 D100 D130  ; 送り現在値
      MRD
      ANI     B302  ; 今回段数ST=1
      D-      D710 R615Z2 Z6
      D-      Z6 D100 D130
      MPP
      D-      R615Z2 D710 Z6
      D+      Z6 D100 D132
      MPP
      DMOV    R685Z2 D230  ; ﾋﾈﾘ自動設定移動角度
      MPS
      AND     L126  ; 終振自動演算有_TB
      AND     B2B4  ; 終点ﾌﾗﾝｼﾞﾗﾝﾌﾟ
      LD      L102  ; 半自動選択_TB
      OR      L100  ; 自動選択_TB
      ANB
      AND     B302  ; 今回段数ST=1
      LDD<>   K0 R20242  ; 捻り_終振
      ORI     M9994  ; 終振り追加
      ANB
      ANI     M9994  ; 終振り追加
      DMOV    R20242 D230
      MPP
      DMOV    R755Z2 D330  ; 曲げ自動設定角度
      DMOV    R687Z2 D232  ; ﾋﾈﾘBn+1設定移動角度
